// TwinCAT 3 PLC project PLC_Convert
// ProgramVersion: 3.1.4026.19
// libraries:
//   Tc2_Database, * (Beckhoff Automation GmbH)
//   Tc2_Drive, * (Beckhoff Automation GmbH)
//   Tc2_EtherCAT, * (Beckhoff Automation GmbH)
//   Tc2_IoFunctions, * (Beckhoff Automation GmbH)
//   Tc2_Math, * (Beckhoff Automation GmbH)
//   Tc2_MC2, * (Beckhoff Automation GmbH)
//   Tc2_MC2_Drive, * (Beckhoff Automation GmbH)
//   Tc2_SerialCom, * (Beckhoff Automation GmbH)
//   Tc2_Standard, * (Beckhoff Automation GmbH)
//   Tc2_System, * (Beckhoff Automation GmbH)
//   Tc2_SystemCX, * (Beckhoff Automation GmbH)
//   Tc2_TcpIp, * (Beckhoff Automation GmbH)
//   Tc2_Utilities, * (Beckhoff Automation GmbH)
//   Tc2_XmlDataSrv, * (Beckhoff Automation GmbH)
//   Tc3_EventLogger, * (Beckhoff Automation GmbH)
//   Tc3_Module, * (Beckhoff Automation GmbH)
//   TcUnit, * (www.tcunit.org)
// project tree:
//   / Control_Task.TcTTO, xFast_Task.TcTTO, Fast_Task.TcTTO, Accessory_Task.TcTTO, TcUnit_Task.TcTTO
//   Data types/METS/ADS Symobol/ E_SYMBOL_AccessState.TcDUT, E_SYMBOL_AdsStates.TcDUT, ST_SYMBOL_AddressInfo.TcDUT
//   Data types/METS/AI Codes And Validation/ E_CodeAI.TcDUT (not stored), E_CodeAIType.TcDUT, E_CodeType.TcDUT, ST_CodeInfo.TcDUT, ST_CodeValidation.TcDUT, ST_RejectItems.TcDUT, ST_RejectReasonsForCase.TcDUT, ST_RejectReasonsForOuter.TcDUT, ST_RejectReasonsForPack.TcDUT
//   Data types/METS/AI Codes And Validation/GS1_Standard/ E_GS1_CodeAIType.TcDUT, E_GS1_CodeLvl.TcDUT, ST_GS1_AI_Attributs.TcDUT, ST_GS1_AI_Definition.TcDUT, ST_GS1_CodeInfo.TcDUT, ST_GS1_CodeValidation.TcDUT, ST_GS1_Decode_AI.TcDUT
//   Data types/METS/Alarms/ E_MessageID.TcDUT, E_MessageType.TcDUT (not stored), ST_AlarmDB.TcDUT (not stored), ST_Alarms.TcDUT, ST_AlarmSettings.TcDUT, ST_AlarmsTable.TcDUT, ST_AlarmStatus.TcDUT, ST_ALARM_Aux.TcDUT
//   Data types/METS/Aliases/ T_CAC_Filename.TcDUT, T_CASE_Barcode.TcDUT, T_Char.TcDUT, T_CHM_Filename.TcDUT, T_CodeBATCH.TcDUT, T_CodeBRAND.TcDUT, T_CodeCRYPTO.TcDUT, T_CodeGTIN.TcDUT (not stored), T_CodeMRP.TcDUT, T_CodePIT.TcDUT, T_CodePO.TcDUT, T_CodePRODUCEDATE.TcDUT, T_CodeRSKU.TcDUT, T_CodeURL.TcDUT, T_DB_LongSTRING.TcDUT, T_FileExtension.TcDUT, T_FolderName.TcDUT, T_FolderPath.TcDUT (not stored), T_FSS_RejecCode.TcDUT, T_HMI_PACK_Barcode.TcDUT, T_ISO8601Time.TcDUT, T_LongSTRING.TcDUT, T_OAC_Filename.TcDUT, T_OCV_Filename.TcDUT, T_OHM_Filename.TcDUT, T_OUTER_Barcode.TcDUT, T_PACK_Barcode.TcDUT, T_PCM_Filename.TcDUT, T_PositiveINT.TcDUT (not stored), T_PositiveDINT.TcDUT (not stored), T_ProductDescription.TcDUT, T_RejectCode.TcDUT, T_TimeLog.TcDUT
//   Data types/METS/Case/CAC/ E_CAC_State.TcDUT, ST_CAC_Data.TcDUT
//   Data types/METS/Case/CHM/CHM Data Structure/GenericHierarchy/Case Item Structures/ ST_CaseContent.TcDUT (not stored), ST_CaseIdentity.TcDUT (not stored), ST_CaseItem.TcDUT (not stored)
//   Data types/METS/Case/CHM/CHM Data Structure/GenericHierarchy/Outer Item Structures/ ST_OuterContent.TcDUT (not stored), ST_OuterIdentity.TcDUT (not stored), ST_OuterItem.TcDUT (not stored)
//   Data types/METS/Case/CHM/CHM Data Structure/GenericHierarchy/Pack Item Structures/ ST_PackIdentity.TcDUT (not stored), ST_PackItem.TcDUT (not stored)
//   Data types/METS/Case/CHM/CHM Data Structure/GenericHierarchy/ ST_DefaultIdentity.TcDUT (not stored)
//   Data types/METS/Case/CHM/CHM Data Structure/ ST_Attributes.TcDUT, ST_CHM_GenericHierarchy.TcDUT (excluded from build), ST_GenericHierarchy.TcDUT, ST_MessageHeader.TcDUT
//   Data types/METS/Case/CHM/ E_CHM_GeneratorState.TcDUT, E_CHM_State.TcDUT, E_CHM_WriteMode.TcDUT (excluded from build), ST_CHM_Data.TcDUT
//   Data types/METS/Case/ E_CASE_State.TcDUT, ST_CasePackerInfo.TcDUT, ST_CASE_CaseQueue.TcDUT, ST_CASE_DefferOuter.TcDUT, ST_CASE_InfeedQueue.TcDUT (not stored), ST_CASE_OperationData.TcDUT
//   Data types/METS/Case/ORCA/ E_ORCA_State.TcDUT, ST_ORCA_BrandInfo.TcDUT, ST_ORCA_Data.TcDUT, ST_ORCA_Outers.TcDUT, ST_ORCA_ProductInfo.TcDUT, ST_ORCA_SiteInfo.TcDUT
//   Data types/METS/Device/CX Unit/Device/ E_CX_DeviceState.TcDUT (not stored)
//   Data types/METS/Device/CX Unit/EtherCAT/ E_CX_EtherCATState.TcDUT, ST_CX_EtherCATDeviceState.TcDUT, ST_CX_EtherCATMasterPNetState.TcDUT, ST_CX_EtherCATMasterState.TcDUT
//   Data types/METS/Device/CX Unit/EtherCAT/Terminal FBs/EBUS/ ST_EBUS_AnalogueDataIn.TcDUT (not stored), ST_EBUS_EtherCATState.TcDUT (not stored)
//   Data types/METS/Device/CX Unit/EtherCAT/Terminal FBs/KBUS/ E_KBUS_RegisterAccessState.TcDUT (not stored), ST_KBUS_AnalogueDataIn.TcDUT (not stored), ST_KBUS_AnalogueDataOut.TcDUT (not stored), ST_KBUS_KL1501DataIn.TcDUT (not stored), ST_KBUS_KL1501DataOut.TcDUT (not stored), ST_KBUS_KL5001Config.TcDUT (not stored)
//   Data types/METS/Device/CX Unit/EtherCAT/Terminal FBs/ ST_EtherCATSlaveInfo.TcDUT (not stored), ST_EtherCATStatus.TcDUT (not stored)
//   Data types/METS/Device/CX Unit/Network/ E_CX_NetworkInfoState.TcDUT (not stored), E_CX_SetAMSNetIDState.TcDUT (not stored), ST_CX_AdapterInfo.TcDUT, ST_CX_NetworkInfo.TcDUT
//   Data types/METS/Device/CX Unit/NOVRAM/ E_CX_NVDataCtrlState.TcDUT (not stored), E_CX_NVDataOpMode.TcDUT, E_CX_NVXMLState.TcDUT, ST_CX_AMSAddress.TcDUT, ST_CX_EL6080DataIn.TcDUT, ST_CX_EL6080DataOut.TcDUT, ST_CX_NVDataBlock.TcDUT
//   Data types/METS/Device/CX Unit/System/ E_CX_HWType.TcDUT (not stored), E_CX_State.TcDUT
//   Data types/METS/Device/Cylinders/ E_CYLINDER_Name.TcDUT, E_CYLINDER_Position.TcDUT (not stored), ST_CYLINDER_Config.TcDUT, ST_CYLINDER_Control.TcDUT, ST_CYLINDER_IN.TcDUT, ST_CYLINDER_OUT.TcDUT (not stored), ST_CYLINDER_Status.TcDUT, ST_CYLINDER_TagID.TcDUT
//   Data types/METS/Device/DB/ E_DB_ScanState.TcDUT, ST_DB_CACDataCtrl.TcDUT, ST_DB_OACDataCtrl.TcDUT (not stored), ST_DB_OCVDataCtrl.TcDUT (not stored)
//   Data types/METS/Device/DB/OLD/ ST_DBResult.TcDUT (excluded from build), ST_DB_CACCheckCtrl.TcDUT (excluded from build), ST_DB_Config.TcDUT, ST_DB_OACCheckCtrl.TcDUT (excluded from build), ST_DB_OCVCheckCtrl.TcDUT (excluded from build), ST_DB_PcvCheckCtrl.TcDUT (excluded from build), ST_DB_ReportDBCtrl.TcDUT, ST_DB_ReportResult.TcDUT
//   Data types/METS/Device/Drive/Analog/Config/ ST_AnalogDrive.TcDUT (not stored)
//   Data types/METS/Device/Drive/Analog/ ST_DriveCtrl.TcDUT, ST_PhtcCtrl.TcDUT (excluded from build)
//   Data types/METS/Device/Drive/MC2/Axis Control/ E_AXIS_MotionType.TcDUT (not stored), ST_AXIS_Control.TcDUT (not stored), ST_AXIS_IN.TcDUT (not stored), ST_AXIS_OUT.TcDUT (not stored), ST_AXIS_Status.TcDUT (not stored)
//   Data types/METS/Device/Drive/MC2/Config/ ST_AXIS_Config.TcDUT (not stored)
//   Data types/METS/Device/Drive/MC2/EtherCAT/AX5000 FBs/ ST_AX5000_TouchProbe.TcDUT (not stored)
//   Data types/METS/Device/Drive/MC2/EtherCAT/Encoder FBs/ ST_DeviceAddress.TcDUT (not stored)
//   Data types/METS/Device/Drive/MC2/ E_MC_Name.TcDUT
//   Data types/METS/Device/Drive/MC2/NC Axis/Cam/ E_CAM_Update.TcDUT (not stored)
//   Data types/METS/Device/Drive/MC2/NC Axis/ E_AXIS_CtrlState.TcDUT (not stored), E_TORQUE_Scaling.TcDUT (not stored), ST_AxisCtrlRamps.TcDUT (not stored), ST_DriveStatus.TcDUT (not stored), ST_LatchPosBuffer.TcDUT (not stored), ST_NC_EncDataIn.TcDUT (not stored), ST_NC_EncDataOut.TcDUT (not stored)
//   Data types/METS/Device/Drive/MC2/TempAxis/ ST_AxisHomeStruct.TcDUT (not stored) (excluded from build), ST_AxisMotionStruct.TcDUT (not stored) (excluded from build)
//   Data types/METS/Device/Drive/Profinet/Config/ ST_ProfinetDrive.TcDUT (not stored), ST_ProfinetMasterConfig.TcDUT (not stored)
//   Data types/METS/Device/Drive/Profinet/ E_DRIVE_Name.TcDUT (not stored), ST_PNetMasterStatus.TcDUT
//   Data types/METS/Device/Drive/Profinet/Parameters/ ST_DataPntAdr.TcDUT (not stored), ST_KeyPadDisplay.TcDUT (not stored), ST_Parameter.TcDUT (not stored), ST_ParameterControl.TcDUT (not stored), ST_Parameters.TcDUT (not stored), ST_Value.TcDUT (not stored)
//   Data types/METS/Device/Drive/Profinet/_G120/Drives/ E_DRIVE_DataType.TcDUT (not stored), ST_DRIVE_INPUT.TcDUT (not stored), ST_DRIVE_OUTPUT.TcDUT (not stored), ST_DRIVE_STATUS.TcDUT (not stored), ST_G120_ExtendedIn.TcDUT (not stored), ST_G120_ExtendedOut.TcDUT (not stored), ST_G120_IN.TcDUT (not stored), ST_G120_OUT.TcDUT (not stored), ST_G120_Status.TcDUT (not stored)
//   Data types/METS/Device/Drive/Profinet/_G120/ ST_G120_Control.TcDUT (not stored)
//   Data types/METS/Device/Encoders/CAMS/ ST_AFS60_Cam.TcDUT, ST_AFS60_CamHMi.TcDUT, ST_AFS60_Config.TcDUT, ST_AFS60_Status.TcDUT
//   Data types/METS/Device/Encoders/ E_ENOCDER_Name.TcDUT, ST_ENCODER_IN.TcDUT, ST_ENCODER_OUT.TcDUT (not stored), ST_ENCODER_Status.TcDUT
//   Data types/METS/Device/IO2 Controls/ E_IO2_InputSource.TcDUT (not stored), E_IO2_Type.TcDUT (not stored), ST_IO2_Diagnostic.TcDUT, ST_IO2_InputPLC.TcDUT, ST_IO2_OutputPLC.TcDUT
//   Data types/METS/Device/IO2 Controls/Input Ctrl/ ST_IO2_DoubleInputCtrl.TcDUT, ST_IO2_DoubleInputLockedCtrl.TcDUT, ST_IO2_SingleInputCtrl.TcDUT, ST_IO2_SingleInputLockedCtrl.TcDUT
//   Data types/METS/Device/IO2 Controls/Outpout Ctrl/ ST_IO2_OutputCtrl.TcDUT
//   Data types/METS/Device/Printers/ E_PRINTER_Name.TcDUT, E_PRINTER_State.TcDUT (not stored), ST_PRINTER_Config.TcDUT, ST_PRINTER_IN.TcDUT, ST_PRINTER_OUT.TcDUT, ST_PRINTER_Status.TcDUT
//   Data types/METS/Device/Scanner/ E_ClientSteps.TcDUT, E_DataExchaSteps.TcDUT, E_SCANNER_CodeType.TcDUT (not stored), E_SCANNER_DeviceType.TcDUT (not stored), E_SCANNER_Name.TcDUT, E_SCANNER_State.TcDUT (not stored), E_SCANNER_Vendor.TcDUT (not stored), ST_SCANNER.TcDUT, ST_SCANNER_ApplicationIdentifier.TcDUT, ST_SCANNER_CameraMap.TcDUT, ST_SCANNER_CodeData.TcDUT, ST_SCANNER_Config.TcDUT, ST_SCANNER_Evaluation.TcDUT, ST_SCANNER_ImageData.TcDUT, ST_SCANNER_ManualCtrl.TcDUT, ST_SCANNER_OpState.TcDUT, ST_SCANNER_Options.TcDUT, ST_SCANNER_Performance.TcDUT, ST_SCANNER_Statistics.TcDUT, ST_SCANNER_TriggerID.TcDUT
//   Data types/METS/Device/Scanner/Hand Scanner/ E_ConnectSteps.TcDUT, E_DataSequence.TcDUT (not stored), E_SCANNER_Baudrate.TcDUT, ST_SCANNER_HoneywellConfig.TcDUT, ST_SCANNER_HoneywellCtrl.TcDUT, ST_SCANNER_HoneywellStatus.TcDUT, ST_SCANNER_HostAck.TcDUT, ST_SCANNER_USBConfig.TcDUT
//   Data types/METS/Device/Scanner/NewModel/ ST_SCANNER_CtrlMapping.TcDUT, ST_SCANNER_Configuration.TcDUT, ST_SCANNER_Ctrl.TcDUT (not stored), ST_SCANNER_IN.TcDUT (not stored), ST_SCANNER_CtrlOptions.TcDUT (not stored) (excluded from build), ST_SCANNER_ManualStatus.TcDUT, ST_SCANNER_OUT.TcDUT, ST_SCANNER_Status.TcDUT
//   Data types/METS/Files/ E_FILE_CtrlState.TcDUT, E_FILE_DeleteOldFilesState.TcDUT, E_FILE_State.TcDUT, ST_FILE_WriteFileStatistic.TcDUT
//   Data types/METS/HMI/Device Manual Control/ ST_HMI_AxisCtrl.TcDUT, ST_HMI_CylinderCtrl.TcDUT, ST_HMI_G120Ctrl.TcDUT, ST_HMI_PrinterCtrl.TcDUT
//   Data types/METS/HMI/Device Status/ E_HMI_DriveStatus.TcDUT, ST_HMI_AxisStatus.TcDUT (not stored), ST_HMI_CylinderStatus.TcDUT, ST_HMI_G120Status.TcDUT, ST_HMI_HoneywellStatus.TcDUT, ST_HMI_PrinterStatus.TcDUT
//   Data types/METS/HMI/HMIQueue/ ST_HMI_CAC_Data.TcDUT, ST_HMI_CaseRejectCode.TcDUT, ST_HMI_CaseVerifiedCode.TcDUT (not stored), ST_HMI_CASE_CaseQueue.TcDUT (not stored), ST_HMI_InfeedQueue.TcDUT, ST_HMI_OAC_Data.TcDUT (not stored), ST_HMI_OCV_Data.TcDUT (not stored), ST_HMI_OuterStatus.TcDUT (not stored), ST_HMI_PACK_BufferStatus.TcDUT, ST_HMI_PLAS_Queue.TcDUT (not stored)
//   Data types/METS/HMI/ ST_HMI_BarGraph.TcDUT, ST_HMI_Buttons.TcDUT, ST_HMI_CSVStoreTable.TcDUT, ST_HMI_StationStatus.TcDUT (not stored), ST_HMI_Visualisation.TcDUT
//   Data types/METS/KPI/ ST_KPI_CasePackerSignals.TcDUT (not stored), ST_KPI_CodePos.TcDUT, ST_KPI_InspectionEfficency.TcDUT, ST_KPI_ItemsProduced.TcDUT, ST_KPI_OCVFile.TcDUT (not stored), ST_KPI_OutersProcessing.TcDUT, ST_KPI_OutersProduced.TcDUT
//   Data types/METS/LogData/ E_LOG_Handler.TcDUT, ST_LOG_Alarms.TcDUT (not stored), ST_LOG_EventData.TcDUT (not stored), ST_LOG_FileWriteError.TcDUT (not stored), ST_LOG_MachineState.TcDUT (not stored), ST_LOG_RejectReasons.TcDUT, ST_LOG_WriteImageData.TcDUT (not stored)
//   Data types/METS/NV Data/ ST_NOVRAM_METS_Cameras.TcDUT, ST_NOVRAM_METS_CaseInspactionLog.TcDUT (not stored), ST_NOVRAM_METS_DualInputs.TcDUT, ST_NOVRAM_METS_EventCounters.TcDUT, ST_NOVRAM_METS_Inspection.TcDUT
//   Data types/METS/Outers/ E_OUTER_AgrregationState.TcDUT, E_OUTER_State.TcDUT, ST_OUTER_Status.TcDUT
//   Data types/METS/Outers/OAC/ E_OAC_State.TcDUT, ST_OAC_Data.TcDUT
//   Data types/METS/Outers/SFLX/ E_SIDEFLEX_UnitType.TcDUT, ST_SIDEFLEX_Offset.TcDUT, ST_SIDEFLEX_ProcessData.TcDUT
//   Data types/METS/Packs/ E_OCV_CheckMode.TcDUT, E_OCV_State.TcDUT, E_PACK_FilledInStatus.TcDUT, E_PACK_ReadStep.TcDUT, E_PACK_State.TcDUT, ST_PACK_CodeBuffer.TcDUT, ST_PACK_CodeStatus.TcDUT, ST_PACK_ConfirmationQueue.TcDUT, ST_PACK_Data.TcDUT, ST_PACK_DuplicatesCheck.TcDUT, ST_PACK_InfeedQueue.TcDUT, ST_PACK_InTransferQueue.TcDUT, ST_PACK_LastFilledCodes.TcDUT, ST_PACK_TriggerOffset.TcDUT
//   Data types/METS/Packs/_Lab/ ST_LAB_PackData.TcDUT, ST_LAB_OuterData.TcDUT
//   Data types/METS/PCM/ E_PCM_State.TcDUT, ST_PCM_Data.TcDUT, ST_PCM_Status.TcDUT (not stored)
//   Data types/METS/PCM/PCM_Hierarchy/ProductInformation/Product/ ST_HierarchyData.TcDUT (not stored), ST_HierarchyDataList.TcDUT (not stored)
//   Data types/METS/PCM/PCM_Hierarchy/ProductInformation/Settings/ ST_ToleranceThresholdCS.TcDUT (not stored), ST_ToleranceThresholdOUT.TcDUT (not stored), ST_ToleranceThresholdPK.TcDUT (not stored)
//   Data types/METS/PCM/PCM_Hierarchy/ProductInformation/ ST_PCMProduct.TcDUT, ST_PCMSettings.TcDUT
//   Data types/METS/PCM/PCM_Hierarchy/ ST_PCMMessageHeader.TcDUT, ST_ProductInformation.TcDUT
//   Data types/METS/String Processing/ E_STRING_ExtrMode.TcDUT
//   Data types/METS/System/ E_SYSTEM_CTState.TcDUT, E_SYSTEM_HandScannerBaudrate.TcDUT, E_SYSTEM_ItemType.TcDUT, E_SYSTEM_MachineState.TcDUT (not stored), E_SYSTEM_MaintainFolders.TcDUT (not stored), E_SYSTEM_OSType.TcDUT, ST_SYSTEM_Config.TcDUT, ST_SYSTEM_DateTime.TcDUT, ST_SYSTEM_DeviceState.TcDUT, ST_SYSTEM_Door.TcDUT, ST_SYSTEM_MachineID.TcDUT, ST_SYSTEM_MachineMode.TcDUT, ST_SYSTEM_MachineState.TcDUT, ST_SYSTEM_ProductionLine.TcDUT, ST_SYSTEM_SafetyStatus.TcDUT, ST_SYSTEM_SoftwareVersion.TcDUT
//   Data types/METS/System/Status/ ST_SYSTEM_ArchiveDBStatus.TcDUT, ST_SYSTEM_ReportingDBStatus.TcDUT (not stored), ST_SYSTEM_BridgeStatus.TcDUT (not stored), ST_SYSTEM_LoggerStatus.TcDUT, ST_SYSTEM_MachineStatus.TcDUT (not stored)
//   Data types/METS/System/System Modes/ E_SYSTEM_AutomationMode.TcDUT, E_SYSTEM_OuterAggregationMode.TcDUT, E_SYSTEM_PackAggregationMode.TcDUT (not stored)
//   Data types/METS/TCPIP Address/ E_TCPIP_State.TcDUT, ST_TCPIP_AddressPort.TcDUT
//   Data types/METS/XML Processing/ E_XML_CtrlState.TcDUT, E_XML_GeneratorState.TcDUT, E_XML_WritingMode.TcDUT
//   Data types/METS/_StationOperational/C715 Tempalate Example/ E_04_ElevatorState_C715.TcDUT, E_Axis_C715.TcDUT, E_Cylinder_C715.TcDUT, ST_04_ElevatorSeq_C715.TcDUT, ST_BundleTrackingRegister_C715.TcDUT, ST_CommonStationConfig_C715.TcDUT
//   Data types/METS/_StationOperational/ E_00_StationStateTemplate.TcDUT, ST_00_StationStructTemplate.TcDUT
//   Data types/METS/_StationOperational/Manual Machine/ E_OuterPrintStationState.TcDUT, ST_OuterPrintStationStruct.TcDUT (not stored)
//   Data types/METS/_StationOperational/SeqCtrl/ ST_STATION_Requests.TcDUT, ST_STATION_Status.TcDUT
//   POUs/METS/Common LIB/04_CASE LIB/Case FBs/FinaliseCaseData/ FB_CASE_DuplicatCheck.TcPOU (not stored), FB_CASE_DuplicateUpdateToDB.TcPOU (not stored), FB_CASE_FinaliseData.TcPOU (not stored), FB_CASE_InitialiseData.TcPOU (not stored), FB_CASE_MovePackerToCase.TcPOU (not stored), FB_CASE_ValidateContent.TcPOU (not stored)
//   POUs/METS/Common LIB/07_DEVICE LIB/CommonCX FBs %28Hardware%29/EtherCAT FBs/Obsolete/ FB_CX_EtherCATDevState.TcPOU (not stored) (excluded from build), FB_CX_EtherCATSlaveDiag.TcPOU (not stored) (excluded from build), FB_EtherCAT_Status.TcPOU (not stored) (excluded from build)
//   POUs/METS/Common LIB/07_DEVICE LIB/CommonCX FBs %28Hardware%29/Non-Volatile Data FBs/Obsolete/ FB_CX_NVData_BinaryFile_4K.TcPOU (not stored) (excluded from build), FB_CX_NVData_EL6080_1K.TcPOU (not stored) (excluded from build), FB_CX_NVData_Generic1K.TcPOU (not stored) (excluded from build)
//   POUs/METS/Common LIB/08_SOFTWARE LIB/AI Codes And Validation FBs/ F_CODE_GetItemAI.TcPOU, FB_CODE_ClearCodeInfo.TcPOU, FB_CODE_ValidateExplicitCode.TcPOU (not stored), F_CODE_AssignValToString.TcPOU, F_CODE_AssignValToStringWithPrefix.TcPOU (not stored), F_CODE_GetItem.TcPOU
//   POUs/METS/Common LIB/09_SYSTEM LIB/Alarm/ FB_ALARM_Handler.TcPOU (not stored), FB_ALARM_GroupManagment.TcPOU (not stored), FB_ALARM_LogTable.TcPOU (not stored), FB_ALARM_Message.TcPOU (not stored) (excluded from build), FB_ALARM_OutputDB.TcPOU (not stored) (excluded from build), F_ALARM_SetDefinition.TcPOU (not stored)
//   POUs/METS/Common LIB/09_SYSTEM LIB/ FB_SYSTEM_CoreFolders.TcPOU, FB_SYSTEM_CorePaths.TcPOU, FB_SYSTEM_AverageTimeDiff.TcPOU, FB_SYSTEM_BarcodeType.TcPOU, FB_SYSTEM_DateTime.TcPOU, FB_SYSTEM_HardwareOS.TcPOU, FB_SYSTEM_MachineState.TcPOU, FB_SYSTEM_ProdMonitor.TcPOU, FB_SYSTEM_SearchBarcode.TcPOU, FB_SYSTEM_SeqControl.TcPOU, FB_SYSTEM_ShiftMonitor.TcPOU, FB_SYSTEM_TaskInfo.TcPOU, FB_SYSTEM_ValidateSettings.TcPOU
//   POUs/METS/METS General/01 Control Task %28Process%29/ C13_CheckDuplicatesCACData.TcPOU (not stored), C01_System.TcPOU (not stored), C02_PCM.TcPOU (not stored), C03_AlarmMessageControl.TcPOU (not stored), C04_ContolButtons.TcPOU (not stored), C05_MachineStatus.TcPOU (not stored), C06_TowerLamps.TcPOU (not stored), C07_EtherCATDiagnostic.TcPOU (not stored), C08_PulseGenerator.TcPOU (not stored), C09_MaintainFolders.TcPOU (not stored), C10_PackControlOCVData.TcPOU (not stored), C11_OuterControlOACData.TcPOU (not stored), C12_InfeedConvAddOACData.TcPOU (not stored), C20_ProfinetDrivesCtrl.TcPOU (not stored), C21_CamerasCtrl.TcPOU (not stored), C25_MC2AxisDriversCtrl.TcPOU (not stored), C30_DiagnosticHMI.TcPOU (not stored)
//   POUs/METS/METS General/02 Accessory Task %28External%29/ A10_LAB_Duplicat.TcPOU (not stored) (excluded from build), A04_StartupWebHMI.TcPOU (not stored), A01_StartupBridge.TcPOU (not stored), A07_BargraphHMI.TcPOU (not stored), A06_AuxInterface.TcPOU (not stored), A08_CodeInfoCtrl.TcPOU (not stored), A09_CurrentStatistic.TcPOU (not stored), A03_StartupLogger.TcPOU (not stored), A02_StartupArchiveDB.TcPOU (not stored), A05_StartupReportingDB.TcPOU (not stored) (excluded from build)
//   POUs/TcUnit/FB_CASE_ValidateContentTests/ FB_CASE_ValidateContentTests.TcPOU, PRG_CASE_ValidateContentManual.TcPOU
//   POUs/_Exclude/ F13_CaseContentValidation_ORG.TcPOU (excluded from build), FB_CASE_FinaliseCaseData.TcPOU (excluded from build), FB_CASE_ValidateCaseContent.TcPOU (excluded from build), FB_SYSTEM_CheckOS.TcPOU (excluded from build), FB_SYSTEM_CreateFolders.TcPOU (excluded from build), C09_MaintainFolders_OLD.TcPOU (excluded from build), C09_MaintainFolders_ORG.TcPOU (excluded from build), F15_CaseControlCACData_ORG.TcPOU (excluded from build), F21_ContentHandScanner_ORG.TcPOU (excluded from build), F41_EventLoggerPT.TcPOU (excluded from build), F42_EventLoggerML.TcPOU (excluded from build), F43_EventLoggerOT.TcPOU (excluded from build), F44_EventLoggerCT.TcPOU (excluded from build), FB_CASE_AddOACDataLoop.TcPOU (excluded from build), FB_CASE_ShiftCaseQueue_ORG.TcPOU (excluded from build), FB_CHM_ClearArchive.TcPOU (excluded from build), FB_CX_NVData_NOVRAM_4K.TcPOU (excluded from build), FB_MemoryMonitor_32K.TcPOU (excluded from build), FB_MemoryMonitor_4K.TcPOU (excluded from build), FB_OUTER_CompleteDataFromConfirmation.TcPOU (excluded from build), FB_OUTER_CompleteDataFromOCV.TcPOU (excluded from build), FB_OUTER_RefeedOCVFilesWtihError.TcPOU (excluded from build), FB_OUTER_RepairOCVContent.TcPOU (excluded from build), FB_OUTER_WriteOACFileLoop.TcPOU (excluded from build), FB_PACK_DuplicatesPackCodes.TcPOU (excluded from build), FB_PACK_ValidateOCVContent.TcPOU (excluded from build), FB_PACK_WriteOCVFileLoop_v3.TcPOU (excluded from build), FB_T03_MoveDataToOCVStatus_ORG.TcPOU (excluded from build), F_ALARM_SetDefinition_ORG.TcPOU (excluded from build), PRG_LARS_ValidationAsConfirmation_ORG.TcPOU (excluded from build), TestBlock_Check3.TcPOU (excluded from build), TestBlock_Check4.TcPOU (excluded from build)
//   Global Variables/ gMessage.TcGVL, gConstants.TcGVL (not stored), gHMI.TcGVL, CodeAI.TcGVL (not stored), gIOFiltered.TcGVL, gPersistent.TcGVL, gNovRAM.TcGVL
//   Global Variables/InputsOutputsDT/ gCamDevice.TcGVL, IOVarDT_S.TcGVL, IOVarDT_H.TcGVL, _Labs.TcGVL
//   Global Variables/InputsOutputs_CML/ IOVariablesCX_CML.TcGVL (excluded from build), IOVariablesEUCA_CML.TcGVL (excluded from build), IOVariablesPACAN_CML.TcGVL (excluded from build), IOVariablesPAOL_CML.TcGVL (excluded from build), IOVariablesPLAS_CML.TcGVL (excluded from build)
//   Global Variables/InputsOutputs_OC/ IOVariablesCX_OC.TcGVL (excluded from build), IOVariablesEUCA_OC.TcGVL (excluded from build), IOVariablesPAOL_OC.TcGVL (excluded from build), IOVariablesPLAS_OC.TcGVL (excluded from build)
//   Global Variables/InputsOutputs_SFLX/ IOVariablesCX_SFLX.TcGVL (excluded from build), IOVariablesEUCA_SFLX.TcGVL (excluded from build), IOVariablesPAOL_SFLX.TcGVL (excluded from build), IOVariablesPLAS_SFLX.TcGVL (excluded from build)
//   Global Variables/METS/ gDevice.TcGVL, gProcess.TcGVL
//   Global Variables/_VERSION/ _VERSION_CONTROL.TcGVL
//   POUs/METS/Common LIB/01_PACK LIB/OCV FBs/ FB_OCV_FindDB.TcPOU
//   POUs/METS/Common LIB/01_PACK LIB/Pack FBs/ FB_PACK_DuplicatesPackCodesDB.TcPOU, FB_PACK_MoveOuterStatusArray.TcPOU, FB_PACK_WriteOCVLoopDB.TcPOU
//   POUs/METS/Common LIB/01_PACK LIB/Pack FBs/PAOL/2CAM %28METS ONE%29/ FB_2CAM_AddPackCodes.TcPOU (not stored), FB_2CAM_CameraBoxRead.TcPOU (not stored), FB_2CAM_CameraSequenceNo.TcPOU (not stored), FB_2CAM_PackScanners2x5Packs.TcPOU (not stored), FB_2CAM_SelectCameraMap.TcPOU (not stored)
//   POUs/METS/Common LIB/01_PACK LIB/Pack FBs/PAOL/3CAM %28LIGHTBOX%29/ FB_3CAM_AddPackCodes.TcPOU (not stored), FB_3CAM_CameraBoxRead.TcPOU (not stored), FB_3CAM_CameraSequenceNo.TcPOU (not stored), FB_3CAM_PackScanners2x5Packs.TcPOU (not stored), FB_3CAM_PackScanners3x4Packs.TcPOU (not stored), FB_3CAM_PackScanners4x3Packs.TcPOU (not stored), FB_3CAM_SelectCameraMap.TcPOU (not stored)
//   POUs/METS/Common LIB/01_PACK LIB/Pack FBs/PAOL/ FB_PAOL_AddNewTriggerID.TcPOU (not stored), FB_PAOL_InfeedCamerasSync.TcPOU (not stored)
//   POUs/METS/Common LIB/01_PACK LIB/Pack FBs/PLAS/ FB_PLAS_AddInterimCodeToQ.TcPOU (not stored), FB_PLAS_AddNewTriggerID.TcPOU (not stored), FB_PLAS_FillInPackData.TcPOU (not stored), FB_PLAS_FillInPackDataWithCodeType.TcPOU (not stored) (excluded from build), FB_PLAS_InterimShiftQueue.TcPOU (not stored), FB_PLAS_MasterListAddToQueue.TcPOU (not stored), FB_PLAS_MasterListFillInPack.TcPOU (not stored), FB_PLAS_MasterListFillInPackRev.TcPOU (not stored), FB_PLAS_MasterListShiftQueue.TcPOU (not stored)
//   POUs/METS/Common LIB/01_PACK LIB/Pack FBs/PLAS/Type 01 %28CW - GD%29/ FB_T01_Add2PackToInfeedQ.TcPOU (not stored), FB_T01_CompleteOCV.TcPOU (not stored), FB_T01_MovePackToStacker.TcPOU (not stored)
//   POUs/METS/Common LIB/01_PACK LIB/Pack FBs/PLAS/Type 02 %28NCW - GD%29/ FB_T02_Add2PackToInfeedQ.TcPOU (not stored), FB_T02_CompleteOCV.TcPOU (not stored), FB_T02_MovePackToStacker.TcPOU (not stored), FB_T02_PackScanners2x5Packs.TcPOU (not stored) (excluded from build)
//   POUs/METS/Common LIB/01_PACK LIB/Pack FBs/PLAS/Type 03 %28NCW - FOCKE%29/ FB_T03_AddMultiPackToInfeedQ.TcPOU (not stored), FB_T03_CompleteOCV.TcPOU (not stored), FB_T03_MoveDataToOCVStatus.TcPOU (not stored), FB_T03_PackScanners2x5Packs.TcPOU (not stored) (excluded from build), FB_T03_PackScanners5x2Packs.TcPOU (not stored) (excluded from build)
//   POUs/METS/Common LIB/01_PACK LIB/Pack FBs/PLAS/Type 04 %28NCW - FOCKE H%29/ FB_T04_AddMultiPackToInfeedQ.TcPOU (not stored), FB_T04_CompleteOCV.TcPOU (not stored), FB_T04_MoveDataToOCVStatus.TcPOU (not stored)
//   POUs/METS/Common LIB/01_PACK LIB/Pack Functions/ F_PACK_GetRejectReasonFSS.TcPOU, F_PACK_HexToPackCode.TcPOU, F_PACK_ProgNumberMap.TcPOU, F_PACK_ValidateCodeASCII.TcPOU, F_PACK_ValidateHexName.TcPOU, F_PACK_ValidateTimeStamp.TcPOU
//   POUs/METS/Common LIB/02_OUTER LIB/OAC FBs/ FB_OAC_FindDB.TcPOU
//   POUs/METS/Common LIB/02_OUTER LIB/Outer FBs/Complete OCV/ FB_OUTER_CompleteDataFromDB_DoubleCam.TcPOU (not stored), FB_OUTER_CompleteDataFromDB_SingleCam.TcPOU (not stored), FB_OUTER_CompleteDataFromQueue_NoCam.TcPOU (not stored)
//   POUs/METS/Common LIB/02_OUTER LIB/Outer FBs/ FB_OUTER_ArchiveInvalidOuters.TcPOU, FB_OUTER_CheckDuplicateStatus.TcPOU, FB_OUTER_FindErrorOuter.TcPOU, FB_OUTER_InterimCameraOut.TcPOU, FB_OUTER_MasterListUpdate.TcPOU, FB_OUTER_MoveOuterStatus.TcPOU, FB_OUTER_RepairOCVContentDB.TcPOU, FB_OUTER_RestoreOCVDataFromStruct.TcPOU, FB_OUTER_ShiftConfimrCodeQ.TcPOU, FB_OUTER_ValidateOuterForReject.TcPOU, FB_OUTER_ValidationCameraOut.TcPOU, FB_OUTER_WriteErrorTable.TcPOU, FB_OUTER_WriteOACLoopDB.TcPOU
//   POUs/METS/Common LIB/02_OUTER LIB/Outer Functions/ F_OUTER_BarcodeToHex.TcPOU, F_OUTER_GetRejectReasonFSS.TcPOU, F_OUTER_HexToBarcode.TcPOU, F_OUTER_ProgNumberMap.TcPOU
//   POUs/METS/Common LIB/04_CASE LIB/Case FBs/ FB_CASE_AddOACDataDBLoop.TcPOU, FB_CASE_AddOuterToInfeedQ.TcPOU, FB_CASE_AddVerifiedCaseBarcode.TcPOU, FB_CASE_BiuldPackerLogString.TcPOU, FB_CASE_FindAndDeleteOuter.TcPOU, FB_CASE_FindCaseInQueue.TcPOU, FB_CASE_LastRowPoisitionBuffer_v2.TcPOU, FB_CASE_MasterListControl.TcPOU, FB_CASE_MoveFailedCAC.TcPOU, FB_CASE_MoveOutersRowToPacker.TcPOU, FB_CASE_MoveVerifiedCAC.TcPOU, FB_CASE_RestoreDataControl.TcPOU, FB_CASE_ShiftCaseQueue.TcPOU, FB_CASE_ShiftPackerQueue.TcPOU, FB_CASE_ValidatePrintCACData.TcPOU
//   POUs/METS/Common LIB/04_CASE LIB/Case Functons/ F_CASE_AddAIBrackets.TcPOU, F_CASE_BarcodeToCACFilename.TcPOU, F_CASE_ClearCACData.TcPOU, F_CASE_ClearCaseQueue.TcPOU, F_CASE_ClearCurrentPackerData.TcPOU, F_CASE_ClearFailedCaseQueue.TcPOU, F_CASE_ClearInfeedQueue.TcPOU, F_CASE_ClearPackerQueue.TcPOU, F_CASE_GetRejectReasonFSS.TcPOU, F_CASE_GetSKUFromHex.TcPOU (not stored)
//   POUs/METS/Common LIB/04_CASE LIB/Files FBs/CAC FBs/ FB_CAC_RestoreDataFromDB.TcPOU (not stored), FB_CAC_WriteHierachyToDB.TcPOU (not stored)
//   POUs/METS/Common LIB/04_CASE LIB/Files FBs/CHM FBs/ FB_CHM_FindFile.TcPOU (not stored), FB_CHM_MoveToArchive.TcPOU (not stored), FB_CHM_SaveFLG_File.TcPOU (not stored), FB_CHM_WriteFSS3Files.TcPOU (not stored)
//   POUs/METS/Common LIB/04_CASE LIB/Files FBs/CHM FBs/FSS3/ FB_CHM_PopulateDataForFSS3.TcPOU (not stored)
//   POUs/METS/Common LIB/04_CASE LIB/Files FBs/CHM FBs/FSS3/v4/ FB_CHM_BiuldXMLImige_v4.TcPOU (not stored), FB_CHM_HierachyFileGenerator.TcPOU (not stored)
//   POUs/METS/Common LIB/06_KPI LIB/ClearStatistic/ FB_KPI_ClearCameraInspection.TcPOU, FB_KPI_ClearExtCSStatistic.TcPOU, FB_KPI_ClearExtOUTStatistic.TcPOU, FB_KPI_ClearExtPKStatistic.TcPOU, FB_KPI_ClearFrontScreenStatistic.TcPOU, FB_KPI_ClearGeneraStatistic.TcPOU, FB_KPI_ClearInspectionStatistic.TcPOU, FB_KPI_ClearPackOuterInspection.TcPOU (excluded from build)
//   POUs/METS/Common LIB/06_KPI LIB/ItemEfficiency/ FB_KPI_CaseEfficiency.TcPOU, FB_KPI_InterimEfficiency.TcPOU (excluded from build), FB_KPI_OutersEfficiency.TcPOU, FB_KPI_PackEfficiency.TcPOU
//   POUs/METS/Common LIB/06_KPI LIB/ItemEfficiency/Generic/ FB_KPI_GenericEfficiency.TcPOU (not stored)
//   POUs/METS/Common LIB/06_KPI LIB/RejectCounters/ FB_KPI_CaseLevelCounter.TcPOU, FB_KPI_OuterLevelCounter.TcPOU, FB_KPI_PackLevelCounter.TcPOU
//   POUs/METS/Common LIB/07_DEVICE LIB/CommonCX FBs %28Hardware%29/CXDisplay FBs/ FB_CX_CX1100Display.TcPOU (not stored) (excluded from build), FB_CX_CX2100Display.TcPOU (not stored) (excluded from build)
//   POUs/METS/Common LIB/07_DEVICE LIB/CommonCX FBs %28Hardware%29/EtherCAT FBs/ FB_CX_EtherCATStatus.TcPOU (not stored)
//   POUs/METS/Common LIB/07_DEVICE LIB/CommonCX FBs %28Hardware%29/ FB_CX_GetDeviceID.TcPOU (not stored)
//   POUs/METS/Common LIB/07_DEVICE LIB/CommonCX FBs %28Hardware%29/Network FBs/ FB_CX_NetworkInfo.TcPOU (not stored), F_CX_LocalIPAddr.TcPOU (not stored)
//   POUs/METS/Common LIB/07_DEVICE LIB/CommonCX FBs %28Hardware%29/Non-Volatile Data FBs/ FB_CX_NVData_NOVRAM.TcPOU (not stored), FB_CX_NVData_XMLFile.TcPOU (not stored)
//   POUs/METS/Common LIB/07_DEVICE LIB/CommonCX FBs %28Hardware%29/Non-Volatile Data FBs/Internal FBs/ FB_CX_NVData_Transfer.TcPOU (not stored), F_ASCIIWordToByteValue.TcPOU (not stored), F_ByteValueToASCIIWord.TcPOU (not stored)
//   POUs/METS/Common LIB/07_DEVICE LIB/CommonCX FBs %28Hardware%29/Terminal FBs/EBUS/ FB_EBUS_020mASensor.TcPOU (not stored), FB_EBUS_10VSensor.TcPOU (not stored), FB_EBUS_420mASensor.TcPOU (not stored), FB_EBUS_TempSensor.TcPOU (not stored)
//   POUs/METS/Common LIB/07_DEVICE LIB/Cylinders/ FB_Cylinder.TcPOU, FB_CylinderWithMeasur.TcPOU (excluded from build)
//   POUs/METS/Common LIB/07_DEVICE LIB/DB Control/Connection Parameters/ FB_DB_CreateConnectionParams.TcPOU (not stored) (excluded from build)
//   POUs/METS/Common LIB/07_DEVICE LIB/DB Control/_internal/ FB_DBStoredProceduresRecordArrayLoop.TcPOU (not stored) (excluded from build)
//   POUs/METS/Common LIB/07_DEVICE LIB/Door/ FB_DOOR_RejectCtrl.TcPOU (excluded from build)
//   POUs/METS/Common LIB/07_DEVICE LIB/Drives/AX5000 FBs/ FB_MC2_AX5000AxisCtrl.TcPOU (not stored), FB_MC2_AX5000LatchPulse.TcPOU (not stored), FB_MC2_AX5000LatchPulseWidth.TcPOU (not stored), FB_MC2_AX5000Torque.TcPOU (not stored), FB_MC2_AX5000TorqueCtrl.TcPOU (not stored)
//   POUs/METS/Common LIB/07_DEVICE LIB/Drives/AX5000 FBs/Internal FBs/ FB_MC2_AX5000Status.TcPOU (not stored)
//   POUs/METS/Common LIB/07_DEVICE LIB/Drives/Axis Ctrl FBs/ FB_MC2_AbsCtrl.TcPOU (not stored), FB_MC2_BasicAxisCtrl.TcPOU (not stored), FB_MC2_CamCtrl.TcPOU (not stored) (excluded from build), FB_MC2_DigLockCtrl.TcPOU (not stored) (excluded from build), FB_MC2_RelCtrl.TcPOU (not stored), FB_MC2_VeloCtrl.TcPOU (not stored)
//   POUs/METS/Common LIB/07_DEVICE LIB/Drives/Conveyors/ FB_ACTransferControl.TcPOU (not stored) (excluded from build), FB_ConveyorControl.TcPOU (not stored) (excluded from build), FB_ConveyorCtrl.TcPOU (not stored) (excluded from build), FB_DriveAnalog.TcPOU (not stored) (excluded from build), FB_SeparatorCtrl.TcPOU (not stored) (excluded from build)
//   POUs/METS/Common LIB/07_DEVICE LIB/Drives/EL7201 FBs/ FB_MC2_EL7201AxisCtrl.TcPOU (not stored), FB_MC2_EL7201Torque.TcPOU (not stored), FB_MC2_EL7201TorqueCtrl.TcPOU (not stored)
//   POUs/METS/Common LIB/07_DEVICE LIB/Drives/EL7201 FBs/Internal FBs/ FB_MC2_EL7201Status.TcPOU (not stored)
//   POUs/METS/Common LIB/07_DEVICE LIB/Drives/Profinet Drives/Drive Control/ FB_DRIVE_SetControl.TcPOU (not stored), FB_G120Simple_V001.TcPOU (not stored), FB_ResetPulseGenerator.TcPOU (not stored), FB_SafetyResetSequencer.TcPOU (not stored) (excluded from build), F_DRIVE_GetStatus.TcPOU (not stored)
//   POUs/METS/Common LIB/07_DEVICE LIB/Drives/Profinet Drives/Drive Parameters/Function Blocks/ FB_ParameterDisplayWrapper.TcPOU (not stored) (excluded from build), FB_ReadDriveParametersPNET.TcPOU (not stored) (excluded from build), FB_WriteDriveParametersPNET.TcPOU (not stored) (excluded from build)
//   POUs/METS/Common LIB/07_DEVICE LIB/Drives/Profinet Drives/Drive Parameters/Functions/ FC_InitG120ReadPara.TcPOU (not stored) (excluded from build), FC_InitG120ReadWritePara.TcPOU (not stored) (excluded from build), FC_ReturnPointerForType.TcPOU (not stored) (excluded from build), FC_Round.TcPOU (not stored) (excluded from build)
//   POUs/METS/Common LIB/07_DEVICE LIB/Encoders/ FB_ENCODER_AbsValueToPos.TcPOU, FB_ENCODER_CamCtrl.TcPOU (excluded from build), FB_ENCODER_SingleTurn.TcPOU
//   POUs/METS/Common LIB/07_DEVICE LIB/IO2 Controls/ FB_IO2_DoubleInputCtrl.TcPOU, FB_IO2_DoubleInputLockCtrl.TcPOU, FB_IO2_ForceOutputs.TcPOU, FB_IO2_OutputCtrl.TcPOU, FB_IO2_SingleInputCtrl.TcPOU, FB_IO2_SingleInputLockCtrl.TcPOU, FB_IO_ForceOutputs.TcPOU (excluded from build)
//   POUs/METS/Common LIB/07_DEVICE LIB/Printer FBs/Domino/ FB_PRINTER_DominoMSeriesCtrl.TcPOU (not stored), FB_PRINTER_SelectCommand.TcPOU (not stored), F_PRINTER_Outer5Fields.TcPOU (not stored)
//   POUs/METS/Common LIB/07_DEVICE LIB/Scanner FBs %28Camera%29/Additional FBs/ FB_SCANNER_CheckOS.TcPOU (not stored), FB_SCANNER_CodeDiagnostic.TcPOU (not stored) (excluded from build), FB_SCANNER_DiagnosticLog.TcPOU (not stored), FB_SCANNER_DecodeGS1.TcPOU (not stored), FB_SCANNER_Evaluation.TcPOU (not stored), FB_SCANNER_KeyenceBrowse.TcPOU (not stored), FB_SCANNER_KeyenceDecodeImageData.TcPOU (not stored), FB_SCANNER_MICROSCANBrowse.TcPOU (not stored), FB_SCANNER_MicroscanDecodeImageData.TcPOU (not stored), FB_SCANNER_MV4x0Browse.TcPOU (not stored), FB_SCANNER_MVxDecodeImageData.TcPOU (not stored), FB_SCANNER_OmronDecodeImageData.TcPOU (not stored), FB_SCANNER_SiemensMV4x0Ctrl_Server.TcPOU (not stored) (excluded from build), F_SCANNER_CodeMaxLenghtCheck.TcPOU (not stored), F_SCANNER_FindCodeType.TcPOU (not stored), F_SCANNER_Keyence_SymbolID_To_CodeType.TcPOU (not stored), F_SCANNER_LightingIntensity.TcPOU (not stored), F_SCANNER_MV4x0Options.TcPOU (not stored) (excluded from build), F_SCANNER_OpState.TcPOU (not stored), F_SCANNER_RemoveAIBrackets.TcPOU (not stored), F_SCANNER_TriggerID.TcPOU (not stored)
//   POUs/METS/Common LIB/07_DEVICE LIB/Scanner FBs %28Camera%29/Cameras/ FB_SCANNER_CameraSelect.TcPOU (not stored), FB_SCANNER_MicroScan.TcPOU (not stored), FB_SCANNER_OmronFJCtrl.TcPOU (not stored), FB_SCANNER_SiemensMV4x0Ctrl.TcPOU (not stored)
//   POUs/METS/Common LIB/07_DEVICE LIB/Scanner FBs %28Camera%29/NewModel/ FB_SCANNER_CameraSelectExt.TcPOU (not stored), FB_SCANNER_KeyenceExt.TcPOU (not stored), FB_SCANNER_OmronExt.TcPOU (not stored), FB_SCANNER_SiemensExt.TcPOU (not stored)
//   POUs/METS/Common LIB/07_DEVICE LIB/Scanner FBs %28Camera%29/SerialScanners/ FB_HandScannerAddress.TcPOU (not stored), FB_HandScannerCtrl.TcPOU (not stored), FB_SCANNER_BaudrateMonitor.TcPOU (not stored), FB_SCANNER_HoneyWellControl.TcPOU (not stored), FB_SCANNER_SerialCom_v2.TcPOU (not stored)
//   POUs/METS/Common LIB/08_SOFTWARE LIB/AI GS1 Codes And Validation FBs/ FB_GS1_ClearCodeInfo.TcPOU, FB_GS1_ValidateExplicitCode.TcPOU, F_GS1_GetItem.TcPOU
//   POUs/METS/Common LIB/08_SOFTWARE LIB/Cog Checker FB/CogChecker/ FB_COG_Chek.TcPOU (not stored) (excluded from build), F_CogCheck.TcPOU (not stored) (excluded from build), F_MulMod.TcPOU (not stored) (excluded from build)
//   POUs/METS/Common LIB/08_SOFTWARE LIB/Cog Checker FB/ FB_CogCorrection.TcPOU (excluded from build), F_COG_Checker.TcPOU (excluded from build)
//   POUs/METS/Common LIB/08_SOFTWARE LIB/Counter FBs/ FB_ChangeStateTrig.TcPOU, FB_CTD32.TcPOU, FB_CTU16.TcPOU, FB_CTU32.TcPOU, FB_Incrementer.TcPOU, FB_InWindow.TcPOU
//   POUs/METS/Common LIB/08_SOFTWARE LIB/Debug/ FB_DEBUG_CounterArray.TcPOU
//   POUs/METS/Common LIB/08_SOFTWARE LIB/File FBs/ FB_FILE_ApendWriteByByte.TcPOU, FB_FILE_Compare.TcPOU, FB_FILE_Copy.TcPOU, FB_FILE_CopyByByte.TcPOU, FB_FILE_Delete.TcPOU, FB_FILE_DeleteOldFiles.TcPOU, FB_FILE_GetFileInfo.TcPOU, FB_FILE_GetFileList.TcPOU, FB_FILE_Move.TcPOU, FB_FILE_MoveWithDate.TcPOU, FB_FILE_ReadByByte.TcPOU, FB_FILE_Rename.TcPOU, FB_FILE_WriteByByte.TcPOU, F_FILE_AppendStringToFileName.TcPOU, F_FILE_CompareFileTime.TcPOU, F_FILE_FileTimeToULarge.TcPOU, F_FILE_SetFileExtension.TcPOU, F_FILE_SplitFilename.TcPOU, F_FILE_SplitPath.TcPOU, F_FILE_TIME_GT.TcPOU, F_FILE_ULargeToFileTime.TcPOU
//   POUs/METS/Common LIB/08_SOFTWARE LIB/IP Address FBs/ F_IP_AddressPort.TcPOU
//   POUs/METS/Common LIB/08_SOFTWARE LIB/Logger FBs/ FB_LOG_FileWriteError.TcPOU, FB_LOG_Handler.TcPOU
//   POUs/METS/Common LIB/08_SOFTWARE LIB/Maths FBs/ FB_CumulativeAverage.TcPOU, FB_Interval.TcPOU, FB_MovingAverage.TcPOU, FB_MovingAverageEvent.TcPOU, FB_MovingAverageTimer.TcPOU, FB_MovingWindowEvent.TcPOU, FB_MovingWindowTimer.TcPOU, F_ApplyTimeOffset.TcPOU, F_CompareSign.TcPOU, F_FileTimeToULarge.TcPOU, F_GetSign.TcPOU, F_Interpolate.TcPOU, F_ModuloPos.TcPOU, F_SafeDIV.TcPOU, F_ULargeToFileTime.TcPOU
//   POUs/METS/Common LIB/08_SOFTWARE LIB/Memory FBs/ FB_StructureMonitor.TcPOU, F_8BitsToByte.TcPOU, F_Checksum_CRC16.TcPOU, F_FiltredSetBitState16.TcPOU (not stored), F_GetBitState.TcPOU, F_PointerToByteADD.TcPOU, F_PointerToWordADD.TcPOU, F_SafeTo_UDINT.TcPOU, F_SetBitState.TcPOU
//   POUs/METS/Common LIB/08_SOFTWARE LIB/String FBs/Concat Function/ F_CONCAT3.TcPOU (not stored), F_CONCAT4.TcPOU (not stored), F_CONCAT5.TcPOU (not stored), F_CONCAT6.TcPOU (not stored), F_CONCAT7.TcPOU (not stored), F_CONCAT8.TcPOU (not stored), F_CONCAT9.TcPOU (not stored)
//   POUs/METS/Common LIB/08_SOFTWARE LIB/String FBs/ FB_ExtractAnyString.TcPOU, FB_ExtractLongString.TcPOU, FB_ExtractString.TcPOU, FB_ExtractString_v2.TcPOU (excluded from build), F_AddPadding.TcPOU, F_AddPaddingUDINT.TcPOU, F_CodeToHex.TcPOU, F_InvalidateASCIIChar.TcPOU, F_InvalidNumericChar.TcPOU, F_IsNumber.TcPOU, F_ReplaceLongSingleChar.TcPOU, F_ReplaceSingleChar.TcPOU, F_ReplaceLongSingleChar.TcPOU, F_StringAddPrefix.TcPOU, F_StringAddSuffix.TcPOU, F_StringWildcard.TcPOU (not stored), F_ValidateString.TcPOU, F_ValidateString_Code.TcPOU, F_WriteEscapeCharacters.TcPOU, F_ZeroPadString.TcPOU
//   POUs/METS/Common LIB/08_SOFTWARE LIB/String FBs/LongConcat Function/ F_LongCONCAT.TcPOU (not stored) (excluded from build), F_LongDELETE.TcPOU (not stored) (excluded from build), F_LongFIND.TcPOU (not stored) (excluded from build), F_LongLEFT.TcPOU (not stored) (excluded from build), F_LongMID.TcPOU (not stored) (excluded from build), F_LongRIGHT.TcPOU (not stored) (excluded from build), F_LongToLowCase.TcPOU (not stored) (excluded from build)
//   POUs/METS/Common LIB/08_SOFTWARE LIB/TcChecks/ CheckBounds.TcPOU (not stored) (excluded from build), CheckDivReal.TcPOU (not stored) (excluded from build), CheckRangeSigned.TcPOU (not stored), CheckRangeUnsigned.TcPOU (not stored)
//   POUs/METS/Common LIB/08_SOFTWARE LIB/TCP FBs/ FB_TCP_ClientPortCtrl.TcPOU, FB_TCP_ClientPortCtrl_V2.TcPOU (not stored), FB_TCP_CloseAllPorts.TcPOU (not stored), FB_TCP_ReceiveData_V2.TcPOU (not stored), FB_TCP_ReceiveLongString.TcPOU (not stored), FB_TCP_ReceiveString.TcPOU (not stored), FB_TCP_SendData.TcPOU (not stored), FB_TCP_ServerPortCtrl.TcPOU (not stored)
//   POUs/METS/Common LIB/08_SOFTWARE LIB/Timer FBs/ FB_Blink.TcPOU (not stored), FB_Debounce.TcPOU (not stored), FB_EventRate.TcPOU (not stored), FB_EventsPerHour.TcPOU (not stored), FB_LongShortPress.TcPOU (not stored), FB_Puls.TcPOU (not stored), FB_PulseGenerator.TcPOU (not stored), FB_PulseGenerator_Sync.TcPOU (not stored), FB_PulseTrain.TcPOU (not stored), FB_SignalDelay.TcPOU (not stored), FB_Slew.TcPOU (not stored), FB_SquareWave.TcPOU (not stored), FB_SquareWave_Sync.TcPOU (not stored), FB_StopWatch.TcPOU (not stored), FB_StopWatch_LREAL.TcPOU (not stored), FB_TaskTime.TcPOU (not stored) (excluded from build), FB_TimeDistance.TcPOU (not stored), FB_TOFR.TcPOU (not stored), FB_TONR.TcPOU (not stored), P_Puls.TcPOU (not stored)
//   POUs/METS/Common LIB/09_SYSTEM LIB/ClearQueue/ FB_SYSTEM_ClearCameraStatus.TcPOU (not stored), FB_SYSTEM_ClearCaseDataArray.TcPOU (not stored), FB_SYSTEM_ClearCasePackerArray.TcPOU (not stored), FB_SYSTEM_ClearHMIQueue.TcPOU (not stored), FB_SYSTEM_ClearMasterListArray.TcPOU (not stored), FB_SYSTEM_ClearOuterArray.TcPOU (not stored), FB_SYSTEM_ClearPackArray.TcPOU (not stored)
//   POUs/METS/Common LIB/09_SYSTEM LIB/PCM FB%27s/ FB_PCM_ReadFile.TcPOU (not stored), FB_PCM_SetData.TcPOU (not stored), FB_PCM_TrackingModeDecode.TcPOU (not stored), FB_PCM_Validate.TcPOU (not stored), FB_PCM_WriteFile.TcPOU (not stored)
//   POUs/METS/Common LIB/09_SYSTEM LIB/System Function/ F_SYSTEM_BoolToBArcodeType.TcPOU (not stored), F_SYSTEM_CameraMonitor.TcPOU (not stored), F_SYSTEM_DriverMonitor.TcPOU (not stored)
//   POUs/METS/Common LIB/09_SYSTEM LIB/System Time Function/ F_SYSTEM_ApplyTimeOffset.TcPOU (not stored), F_SYSTEM_Date.TcPOU (not stored), F_SYSTEM_DateCodeToDate.TcPOU (not stored), F_SYSTEM_DateCompare.TcPOU (not stored), F_SYSTEM_DateToDateCode.TcPOU (not stored), F_SYSTEM_DayOfYear.TcPOU (not stored), F_SYSTEM_DaysIntToTime.TcPOU (not stored), F_SYSTEM_HMIDateTime.TcPOU (not stored), F_SYSTEM_HMIDateTime_V2.TcPOU (not stored), F_SYSTEM_StringToTime.TcPOU (not stored), F_SYSTEM_SystemTimeAsISO8601.TcPOU (not stored), F_SYSTEM_SystemTimeOffsetToHHMM.TcPOU (not stored), F_SYSTEM_SystemTimeToCHM_Header.TcPOU (not stored), F_SYSTEM_SystemTimeToFolderName.TcPOU (not stored), F_SYSTEM_SystemTimeToOHMFolderName.TcPOU (not stored), F_SYSTEM_Time.TcPOU (not stored), F_SYSTEM_TimeFine.TcPOU (not stored), F_SYSTEM_TimeSuperFine.TcPOU (not stored), F_SYSTEM_ValidProduceDate.TcPOU (not stored)
//   POUs/METS/Common LIB/10_SIMULATOR LIB/Code Generator/ C91_FB_CharacterGenerator.TcPOU (not stored), C91_FB_OuterCodeAggregator.TcPOU (not stored), C91_FB_OuterCodeGenerator.TcPOU (not stored), C91_FB_PackCodeAggregator.TcPOU (not stored), C91_FB_PackCodeGenerator.TcPOU (not stored)
//   POUs/METS/Common LIB/10_SIMULATOR LIB/Code Generator/Code Generator/FB - Not used/ FB_CODE_BATSerializator.TcPOU (not stored)
//   POUs/METS/Common LIB/10_SIMULATOR LIB/Code Generator/Code Generator/ FB_CODE_CaseCodeGenerator.TcPOU (not stored), FB_CODE_OuterCodeGenerator.TcPOU (not stored), F_CODE_BATSerializator.TcPOU (not stored)
//   POUs/METS/Common LIB/10_SIMULATOR LIB/Code Generator/OLD/ C90_FB_CaseCodeGenerator.TcPOU (not stored) (excluded from build), C90_FB_CharacterGenerator.TcPOU (not stored) (excluded from build), C90_FB_Codes_Aggregator.TcPOU (not stored) (excluded from build), C90_FB_PackCodeGenerator.TcPOU (not stored) (excluded from build), C90_Generator.TcPOU (not stored) (excluded from build)
//   POUs/METS/METS General/00 Fast Task %28Devices%29/Automation Mode/CML SEQUENCE/ PRG_CML_01_InfeedCtrl.TcPOU (not stored), PRG_CML_02_LoweratorCtrl.TcPOU (not stored), PRG_CML_03_AdditionalConvCtrl.TcPOU (not stored) (excluded from build)
//   POUs/METS/METS General/00 Fast Task %28Devices%29/Automation Mode/LARS SEQUENCE/ PRG_LARS_01_TransportConvCtrl.TcPOU (not stored), PRG_LARS_02_GateSeparationCtrl.TcPOU (not stored), PRG_LARS_03_AddtitionalConvCtrl.TcPOU (not stored)
//   POUs/METS/METS General/00 Fast Task %28Devices%29/Automation Mode/SFLX SEQUENCE/ PRG_SFLX_01_TransportConvCtrl.TcPOU (not stored), PRG_SFLX_02_OutfeedConvCtrl.TcPOU (not stored), PRG_SFLX_03_AddtitionalConvCtrl.TcPOU (not stored)
//   POUs/METS/METS General/00 Fast Task %28Devices%29/ F00_Safety_Signals.TcPOU (not stored), F01_METS_SingleInputs.TcPOU (not stored), F02_METS_DoubleInputs.TcPOU (not stored), F04_PackAggrergationCtrl.TcPOU (not stored), F06_OuterAutomationCtrl.TcPOU (not stored), F08_OuterAggregationCtrl.TcPOU (not stored), F10_CasePackerDoorCtrl.TcPOU (not stored), F11_InfeedConvQueueCtrl.TcPOU (not stored), F11_InfeedConvQueueCtrl_V3.TcPOU (not stored) (excluded from build), F12_PackerQueuesCtrl.TcPOU (not stored), F13_CaseContentValidation.TcPOU (not stored), F14_CaseQueueControl.TcPOU (not stored), F15_CaseControlCACData.TcPOU (not stored), F18_ClearSystemQueues.TcPOU (not stored), F19_ClearInspectionStatistic.TcPOU (not stored), F20_HandScanner.TcPOU (not stored), F21_ContentHandScanner.TcPOU (not stored), F22_AggregationHandScanner.TcPOU (not stored), F25_CylindersCtrl.TcPOU (not stored), F26_EncodersCtrl.TcPOU (not stored), F30_PrintersCommCtrl.TcPOU (not stored), F32_InterimPrinter.TcPOU (not stored), F33_OuterPrinters.TcPOU (not stored), F33_OuterPrinters_v2_Evo.TcPOU (not stored) (excluded from build), F34_CasePrinter.TcPOU (not stored), F40_StationManager.TcPOU (not stored), F45_EventLoggerExt.TcPOU (not stored), F60_METS_Outputs.TcPOU (not stored), F95_CameraTest.TcPOU (not stored), F96_CHMTester.TcPOU (not stored) (excluded from build), F97_CodesGenerator.TcPOU (not stored) (excluded from build), F98_TCPServer.TcPOU (not stored) (excluded from build), F99_DiagnosticBlock.TcPOU (not stored)
//   POUs/METS/METS General/00 Fast Task %28Devices%29/Outer Aggregation Mode/CML/ PRG_CML_SynchroAggregation.TcPOU (not stored), PRG_CML_ValidationAsConfirmation.TcPOU (not stored)
//   POUs/METS/METS General/00 Fast Task %28Devices%29/Outer Aggregation Mode/LARS/ PRG_LARS_SynchroAggregation.TcPOU (not stored), PRG_LARS_ValidationAsConfirmation.TcPOU (not stored)
//   POUs/METS/METS General/00 Fast Task %28Devices%29/Outer Aggregation Mode/SFLX/ PRG_SFLX_NoValidationCamera.TcPOU (not stored), PRG_SFLX_ValidationAsConfirmation.TcPOU (not stored)
//   POUs/METS/METS General/00 Fast Task %28Devices%29/Pack Aggregation Mode/PAOL SEQUENCE/2CAM_METSONE/ PRG_PAOL_01_LightboxScanersCtrl.TcPOU (not stored)
//   POUs/METS/METS General/00 Fast Task %28Devices%29/Pack Aggregation Mode/PAOL SEQUENCE/3CAM_LIGHTBOX/ PRG_PAOL_02_LightboxScanersCtrl.TcPOU (not stored), PRG_PAOL_03_LightboxSeparatorCtrl.TcPOU (not stored)
//   POUs/METS/METS General/00 Fast Task %28Devices%29/Pack Aggregation Mode/PLAS SEQUENCE/T01_CW_GD/ PRG_PLAS_01_PrimaryMasterListCtrl.TcPOU (not stored), PRG_PLAS_02_PackAggregationCtrl.TcPOU (not stored), PRG_PLAS_03_PackToStackerCtrl.TcPOU (not stored), PRG_PLAS_04_CompleteOuterCtrl.TcPOU (not stored)
//   POUs/METS/METS General/00 Fast Task %28Devices%29/Pack Aggregation Mode/PLAS SEQUENCE/T02_NCW_GD/ PRG_PLAS_05_PrimaryMasterListCtrl.TcPOU (not stored), PRG_PLAS_06_PackAggregationCtrl.TcPOU (not stored), PRG_PLAS_07_PackToStackerCtrl.TcPOU (not stored), PRG_PLAS_08_InterimCamCtrl.TcPOU (not stored), PRG_PLAS_09_CompleteOuterCtrl.TcPOU (not stored)
//   POUs/METS/METS General/00 Fast Task %28Devices%29/Pack Aggregation Mode/PLAS SEQUENCE/T03_NCW_FOCKE/ PRG_PLAS_10_PrimaryMasterListCtrl.TcPOU (not stored), PRG_PLAS_11_PackAggregationCtrl.TcPOU (not stored), PRG_PLAS_12_MovePacksToOCVCtrl.TcPOU (not stored), PRG_PLAS_13_InterimCamCtrl.TcPOU (not stored), PRG_PLAS_14_CompleteOuterCtrl.TcPOU (not stored)
//   POUs/METS/METS General/00 Fast Task %28Devices%29/Pack Aggregation Mode/PLAS SEQUENCE/T04_NCW_FOCKE_HYBRID/ PRG_PLAS_15_PrimaryMasterListCtrl.TcPOU (not stored), PRG_PLAS_16_PackAggregationCtrl.TcPOU (not stored), PRG_PLAS_17_MovePacksToOCVCtrl.TcPOU (not stored), PRG_PLAS_18_InterimCamCtrl.TcPOU (not stored), PRG_PLAS_19_CompleteOuterCtrl.TcPOU (not stored), PRG_PLAS_20_LightboxSeparatorCtrl.TcPOU (not stored)
//   POUs/METS/METS General/03 xFast Task %28Data Base%29/ X00_TimeLogger.TcPOU (not stored) (excluded from build), X02_Database.TcPOU (not stored) (excluded from build), X03_CyclicReport.TcPOU (not stored) (excluded from build), X10_xFastOutputs.TcPOU (not stored) (excluded from build)
//   POUs/METS/ T00_FAST.TcPOU, T01_CONTROL.TcPOU, T02_ACCESSORY.TcPOU, T03_xFAST.TcPOU
//   POUs/TcUnit/FB_ExtractAnyStringTests/ FB_ExtractAnyStringTests.TcPOU, PRG_ExtractAnyStringManual.TcPOU
//   POUs/TcUnit/FB_ExtractStringTests/ FB_ExtratcStringTests.TcPOU, PRG_ExtractStringManual.TcPOU
//   POUs/TcUnit/FB_LOGHandlerTests/ FB_LogHandlerTests.TcPOU, PRG_LogHandlerManual.TcPOU
//   POUs/TcUnit/FUN_ReplaceLongSingleCharTests/ FB_ReplaceLongStringCharTests.TcPOU, PRG_ReplaceLongSingleCharManual.TcPOU
//   POUs/TcUnit/ PRG_TEST.TcPOU
//   POUs/_Exclude/DUT/ E_LOG_HandlerName_OLD.TcDUT (excluded from build), ST_SYSTEM_Config_old.TcDUT (excluded from build)
//   POUs/_Exclude/FSS2/ FB_FSS2_BuildXMLData.TcPOU (excluded from build), FB_FSS2_BuildXMLDataForGMES.TcPOU (excluded from build), FB_FSS2_WriteFile.TcPOU (excluded from build), FB_FSS2_WriteFileForGMES.TcPOU (excluded from build), FB_FSS2_XMLImageGenerator.TcPOU (excluded from build)
//   POUs/_Exclude/OAC FBs/ FB_OAC_BuildXMLData.TcPOU (excluded from build), FB_OAC_ClearArchive.TcPOU (excluded from build), FB_OAC_FindFile.TcPOU (excluded from build), FB_OAC_WriteFile.TcPOU (excluded from build)
//   POUs/_Exclude/OCV FBs/ FB_OCV_BuildXMLData.TcPOU (excluded from build), FB_OCV_ClearArchive.TcPOU (excluded from build), FB_OCV_FindFile.TcPOU (excluded from build), FB_OCV_FindFileWithError.TcPOU (excluded from build), FB_OCV_WriteFile.TcPOU (excluded from build)
//   POUs/_Exclude/v1/ FB_CAC_MoveToArchive.TcPOU (excluded from build), FB_CAC_PopulateMinimalOuterData.TcPOU (excluded from build), FB_CAC_WriteFile.TcPOU (excluded from build)
//   POUs/_Exclude/v1_1/ FB_CHM_BiuldXMLImige.TcPOU (excluded from build), FB_CHM_XMLImageGenerator.TcPOU (excluded from build)
//   POUs/_Exclude/v2/ FB_CAC_MoveFromArchive.TcPOU (excluded from build), FB_CAC_RestoreOAC.TcPOU (excluded from build), FB_CAC_WriteFile_v2.TcPOU (excluded from build), FB_CAC_WriteToArchive_v2.TcPOU (excluded from build)
//   POUs/_Exclude/v2_1/ FB_CHM_BiuldXMLImige_v2.TcPOU (excluded from build), FB_CHM_HierachyGenerator.TcPOU (excluded from build)
//   POUs/_Exclude/v3/ FB_CHM_BiuldXMLImige_v3.TcPOU (excluded from build)
//   POUs/_Exclude/XML/ FB_CX_NVData_XMLFile_32K.TcPOU (excluded from build), FB_CX_NVData_XMLFile_4K.TcPOU (excluded from build)

CONFIGURATION PLC_Convert
    RESOURCE PLC ON TwinCAT3
        TASK Control_Task(INTERVAL := T#12ms, PRIORITY := 22);
        TASK xFast_Task(INTERVAL := T#1ms, PRIORITY := 20);
        TASK Fast_Task(INTERVAL := T#3ms, PRIORITY := 21);
        TASK Accessory_Task(INTERVAL := T#100000us, PRIORITY := 23);
        TASK TcUnit_Task(INTERVAL := T#10ms, PRIORITY := 25);
        PROGRAM T01_CONTROL WITH Control_Task : T01_CONTROL;
        PROGRAM T03_xFAST WITH xFast_Task : T03_xFAST;
        PROGRAM T00_FAST WITH Fast_Task : T00_FAST;
        PROGRAM T02_ACCESSORY WITH Accessory_Task : T02_ACCESSORY;
        PROGRAM PRG_TEST WITH TcUnit_Task : PRG_TEST;
    END_RESOURCE
END_CONFIGURATION

// ---- Data types/METS/ADS Symobol/E_SYMBOL_AccessState.TcDUT
TYPE E_SYMBOL_AccessState :
(
	E_SYMBOL_IDLE,
	E_SYMBOL_GETSYMBOLINFO,
	E_SYMBOL_READDATA,
	E_SYMBOL_WRITEDATA,
	E_SYMBOL_DONE
);
END_TYPE

// ---- Data types/METS/ADS Symobol/E_SYMBOL_AdsStates.TcDUT
TYPE E_SYMBOL_AdsStates :
(
	ADSSTATES_INVALID :=0,
	ADSSTATES_IDLE :=1,
	ADSSTATES_RESET :=2,
	ADSSTATES_INIT :=3,
	ADSSTATES_START :=4,
	ADSSTATES_RUN :=5,
	ADSSTATES_STOP :=6,
	ADSSTATES_SAVECFG :=7,
	ADSSTATES_LOADCFG :=8,
	ADSSTATES_POWERFAILURE :=9,
	ADSSTATES_POWERGOOD :=10,
	ADSSTATES_ERROR :=11
);
END_TYPE

// ---- Data types/METS/ADS Symobol/ST_SYMBOL_AddressInfo.TcDUT
TYPE ST_SYMBOL_AddressInfo :	(* 8 bytes *)
STRUCT
	pSymAddr	: 	DWORD;
	nSymSize	:	UDINT;
END_STRUCT
END_TYPE

// ---- Data types/METS/AI Codes And Validation/E_CodeAIType.TcDUT
TYPE E_CodeAIType :
STRUCT
	GTIN 			: 	INT := 1;
	BatchID 			: 	INT := 10;
	SerialCode		: 	INT := 21;
	ProductionOrder 	: 	INT := 91;
	CryptoCode		: 	INT := 93;
	RSKU 			: 	INT := 240;
	MRP				:	INT := 8005;
	BrandSpecification 	:	INT := 92;
	ProduceDate		:	INT := 94;
	UserField3		:	INT;
END_STRUCT
END_TYPE

// ---- Data types/METS/AI Codes And Validation/E_CodeType.TcDUT
TYPE E_CodeType :
(
	E_NONE,
	E_PACK,
	E_INTERIM,
	E_OUTER,
	E_CASE

);
END_TYPE

// ---- Data types/METS/AI Codes And Validation/GS1_Standard/E_GS1_CodeAIType.TcDUT
TYPE E_GS1_CodeAIType :
(
	GS1_00		:= 0,		(*GS1 Not defined*)
	GS1_01		 :=1,		(***********Global Trade Item Number (GTIN)	N2+N14*************)
	GS1_10		:=10,		(***********Batch or lot number	N2+X..20*************)
	GS1_11		:=11,		(***********Production date (YYMMDD)		N2+N6*************)
	GS1_15		:=15,		(***********Best before date (YYMMDD)			N2+N6*************)
	GS1_17		:=17,		(***********Expiration date (YYMMDD)		N2+N6*************)
	GS1_21		:=21,		(***********Serial number		N2+X..20*************)
	GS1_240		:=240,	(***********Additional product identification assigned by the manufacturer	N3+X..30*************)
	GS1_8005		:=8005,	(***********Price per unit of measure	N4+N6*************)
	GS1_8006		:=8006,	(***********Identification of an individual trade item piece	N4+N14+N2+N2*************)
	GS1_8008		:=8008,	(***********Date and time of production		N4+N8+N..4*************)
	GS1_91		:=91,		(***********Company internal information	N2+X..90*************)
	GS1_92		:=92,		(***********Company internal information	N2+X..90*************)
	GS1_93		:=93,		(***********Company internal information	N2+X..90*************)
	GS1_94		:=94,		(***********Company internal information	N2+X..90*************)
	NON_GS1_01		:=10001,	(***********Non GS1 - user defined		X..255*************)
	NON_GS1_02		:=10002,	(***********Non GS1 - user defined		X..255*************)
	NON_GS1_03		:=10003,	(***********Non GS1 - user defined		X..255*************)
	NON_GS1_04		:=10004,	(***********Non GS1 - user defined		X..255*************)
	NON_GS1_05		:=10005,	(***********Non GS1 - user defined		X..255*************)
	NON_GS1_06		:=10006,	(***********Non GS1 - user defined		X..255*************)
	NON_GS1_07		:=10007,	(***********Non GS1 - user defined		X..255*************)
	NON_GS1_08		:=10008,	(***********Non GS1 - user defined		X..255*************)
	NON_GS1_09		:=10009,	(***********Non GS1 - user defined		X..255*************)
	NON_GS1_10		:=10010	(***********Non GS1 - user defined		X..255*************)
);
END_TYPE

// ---- Data types/METS/AI Codes And Validation/GS1_Standard/E_GS1_CodeLvl.TcDUT
TYPE E_GS1_CodeLvl :
(
	E_LVL_NONE,
	E_LEVEL1,
	E_LEVEL2,
	E_LEVEL3
);
END_TYPE

// ---- Data types/METS/AI Codes And Validation/GS1_Standard/ST_GS1_AI_Attributs.TcDUT
TYPE ST_GS1_AI_Attributs :
STRUCT
	sDataField 	: T_MaxString;
	bDataChanged	: BOOL;
	sAI_Id		: STRING(5);
	eGS1_AI		: E_GS1_CodeAIType;
	bFixed		: BOOL;
	nLength		: UINT;
END_STRUCT
END_TYPE

// ---- Data types/METS/AI Codes And Validation/GS1_Standard/ST_GS1_AI_Definition.TcDUT
TYPE ST_GS1_AI_Definition :
STRUCT
	sDotCode_CI	: STRING(3) := ']j';			(* GS1 marker (FNC1 Carrier Identifiers for DataMatrix barcode *)
	sDMC_CI		: STRING(3) := ']d2';			(* GS1 marker (FNC1 Carrier Identifiers for DataMatrix barcode *)
	sCode128_CI	: STRING(3) := ']c1';			(* GS1 marker (FNC1 Carrier Identifiers for Code128 barcode *)
	stAI_01_Lvl1	: ST_GS1_AI_Attributs := (sAI_Id:='01', eGS1_AI:=GS1_01, bFixed:= TRUE, nLength:=14);	(***********N2+N14*************)
	stAI_01_Lvl2	: ST_GS1_AI_Attributs := (sAI_Id:='01', eGS1_AI:=GS1_01, bFixed:= TRUE, nLength:=14);	(***********N2+N14*************)
	stAI_01_Lvl3	: ST_GS1_AI_Attributs := (sAI_Id:='01', eGS1_AI:=GS1_01, bFixed:= TRUE, nLength:=14);	(***********N2+N14*************)
	stAI_10		: ST_GS1_AI_Attributs := (sAI_Id:='10', eGS1_AI:=GS1_10, bFixed:= FALSE, nLength:=20);	(***********N2+X..20*************)
	stAI_11		: ST_GS1_AI_Attributs := (sAI_Id:='11', eGS1_AI:=GS1_11, bFixed:= TRUE, nLength:=6);	(***********N2+N6*************)
	stAI_15		: ST_GS1_AI_Attributs := (sAI_Id:='15', eGS1_AI:=GS1_15, bFixed:= TRUE, nLength:=6);	(***********N2+N6*************)
	stAI_17		: ST_GS1_AI_Attributs := (sAI_Id:='17', eGS1_AI:=GS1_17, bFixed:= TRUE, nLength:=6);	(***********N2+N6*************)
	stAI_21		: ST_GS1_AI_Attributs := (sAI_Id:='21', eGS1_AI:=GS1_21, bFixed:= FALSE, nLength:=20);	(***********N2+X..20*************)
	stAI_240		: ST_GS1_AI_Attributs := (sAI_Id:='240', eGS1_AI:=GS1_240, bFixed:= FALSE, nLength:=30);		(***********N3+X..30*************)
	stAI_8005		: ST_GS1_AI_Attributs := (sAI_Id:='8005', eGS1_AI:=GS1_8005, bFixed:= TRUE, nLength:=6);		(***********N4+N6*************)
	stAI_8006		: ST_GS1_AI_Attributs := (sAI_Id:='8006', eGS1_AI:=GS1_8006, bFixed:= TRUE, nLength:=18);	(***********N4+N14+N2+N2*************)
	stAI_8008		: ST_GS1_AI_Attributs := (sAI_Id:='8008', eGS1_AI:=GS1_8008, bFixed:= TRUE, nLength:=12);	(***********N4+N8+N..4*************)
	stAI_91		: ST_GS1_AI_Attributs := (sAI_Id:='91', eGS1_AI:=GS1_91, bFixed:= FALSE, nLength:=90);		(***********N2+X..90*************)
	stAI_92		: ST_GS1_AI_Attributs := (sAI_Id:='92', eGS1_AI:=GS1_92, bFixed:= FALSE, nLength:=90);		(***********N2+X..90*************)
	stAI_93		: ST_GS1_AI_Attributs := (sAI_Id:='93', eGS1_AI:=GS1_93, bFixed:= FALSE, nLength:=90);		(***********N2+X..90*************)
	stAI_94		: ST_GS1_AI_Attributs := (sAI_Id:='94', eGS1_AI:=GS1_94, bFixed:= FALSE, nLength:=90);		(***********N2+X..90*************)

	stNON_GS1_01		: ST_GS1_AI_Attributs := (sAI_Id:='10001', eGS1_AI:=NON_GS1_01, bFixed:= FALSE, nLength:=255);		(***********X..255*************)
	stNON_GS1_02		: ST_GS1_AI_Attributs := (sAI_Id:='10002', eGS1_AI:=NON_GS1_02, bFixed:= FALSE, nLength:=255);		(***********X..255*************)
	stNON_GS1_03		: ST_GS1_AI_Attributs := (sAI_Id:='10003', eGS1_AI:=NON_GS1_03, bFixed:= FALSE, nLength:=255);		(***********X..255*************)
	stNON_GS1_04		: ST_GS1_AI_Attributs := (sAI_Id:='10004', eGS1_AI:=NON_GS1_04, bFixed:= FALSE, nLength:=255);		(***********X..255*************)
	stNON_GS1_05		: ST_GS1_AI_Attributs := (sAI_Id:='10005', eGS1_AI:=NON_GS1_05, bFixed:= FALSE, nLength:=255);		(***********X..255*************)
	stNON_GS1_06		: ST_GS1_AI_Attributs := (sAI_Id:='10006', eGS1_AI:=NON_GS1_06, bFixed:= FALSE, nLength:=255);		(***********X..255*************)
	stNON_GS1_07		: ST_GS1_AI_Attributs := (sAI_Id:='10007', eGS1_AI:=NON_GS1_07, bFixed:= FALSE, nLength:=255);		(***********X..255*************)
	stNON_GS1_08		: ST_GS1_AI_Attributs := (sAI_Id:='10008', eGS1_AI:=NON_GS1_08, bFixed:= FALSE, nLength:=255);		(***********X..255*************)
	stNON_GS1_09		: ST_GS1_AI_Attributs := (sAI_Id:='10009', eGS1_AI:=NON_GS1_09, bFixed:= FALSE, nLength:=255);		(***********X..255*************)
	stNON_GS1_10		: ST_GS1_AI_Attributs := (sAI_Id:='10010', eGS1_AI:=NON_GS1_10, bFixed:= FALSE, nLength:=255);		(***********X..255*************)

END_STRUCT
END_TYPE

// ---- Data types/METS/AI Codes And Validation/GS1_Standard/ST_GS1_CodeInfo.TcDUT
TYPE ST_GS1_CodeInfo :
STRUCT
	eCodeLvlType					:	E_GS1_CodeLvl;

	nMinLength					: 	INT;
	nEntireLength					:	INT;
	bValidateEntireLength			: 	BOOL;
	nNumberOfAIs					:	INT;

	stGS1_Field 					: ARRAY[1..cMAX_VALIDATION_ITEMS] OF 	ST_GS1_CodeValidation	;

	(*stGS1_Field01 				:	ST_GS1_CodeValidation	;
	stGS1_Field02 					:	ST_GS1_CodeValidation	;
	stGS1_Field03 					:	ST_GS1_CodeValidation	;
	stGS1_Field04 					:	ST_GS1_CodeValidation	;
	stGS1_Field05					:	ST_GS1_CodeValidation	;
	stGS1_Field06					:	ST_GS1_CodeValidation	;
	stGS1_Field07		 			:	ST_GS1_CodeValidation	;
	stGS1_Field08					:	ST_GS1_CodeValidation	;
	stGS1_Field09					:	ST_GS1_CodeValidation	;
	stGS1_Field10					:	ST_GS1_CodeValidation	;*)

END_STRUCT
END_TYPE

// ---- Data types/METS/AI Codes And Validation/GS1_Standard/ST_GS1_CodeValidation.TcDUT
TYPE ST_GS1_CodeValidation :
STRUCT

	bValidate 			:	BOOL;
	sFieldName		:	STRING(15)	:='';

	sStartAI 			: 	STRING(6)		:= '';
	sEndAI 			: 	STRING(6) 	:= '';
	nCodeStartPos		:	INT;
	nCodeLength		:	INT;

	eGS1_AIType		: 	E_GS1_CodeAIType 	:= GS1_00;

(* If sStartAI is empty, then use nCodeStartPos, else find sStartAI in code for start position *)
(* If sEndAI is empty then use nCodeLength, else find sEndAI in code for end position*)

(*General Application Idendifiers (AI) Description:
	01:		GTIN
	10: 		Batch ID/WorkOrderID
	21: 		Serial Code
	91:		Production Order/WorkCenterID
	93:		Crypto
	240:		RSKU
*)

END_STRUCT
END_TYPE

// ---- Data types/METS/AI Codes And Validation/GS1_Standard/ST_GS1_Decode_AI.TcDUT
TYPE ST_GS1_Decode_AI :
STRUCT
	sAI_Id		: STRING(5);
	bFixed		: BOOL;
	nLength		: UINT;
END_STRUCT
END_TYPE

// ---- Data types/METS/AI Codes And Validation/ST_CodeInfo.TcDUT
TYPE ST_CodeInfo :
STRUCT
	eCodeType					:	E_CodeType;

	nMinLength					: 	INT;
	nEntireLength					:	INT;
	bValidateEntireLength			: 	BOOL;
	nNumberOfAIs					:	INT;

	stGTIN 						:	ST_CodeValidation	:=		(sFieldName :='GTIN',						bNameEditable := FALSE, 		nGS1_AI := 1);
	stBatchID 						:	ST_CodeValidation	:=		(sFieldName :='BatchID', 				bNameEditable := FALSE, 		nGS1_AI := 10);
	stSerialCode 					:	ST_CodeValidation	:=		(sFieldName :='SerialCode', 			bNameEditable := FALSE, 		nGS1_AI := 21);
	stProductionOrder 				:	ST_CodeValidation	:=		(sFieldName :='ProductionOrder', 		bNameEditable := FALSE, 		nGS1_AI := 91);
	stCryptoCode					:	ST_CodeValidation	:=		(sFieldName :='CryptoCode', 			bNameEditable := FALSE, 		nGS1_AI := 93);
	stRSKU						:	ST_CodeValidation	:=		(sFieldName :='RSKU', 						bNameEditable := FALSE, 		nGS1_AI := 240);
	stMRP		 				:	ST_CodeValidation	:=		(sFieldName :='MRP', 						bNameEditable := FALSE, 		nGS1_AI := 8005);
	stBrandSpecification			:	ST_CodeValidation	:=		(sFieldName :='BrandSpec',			bNameEditable := FALSE, 		nGS1_AI := 92);
	stProduceDate					:	ST_CodeValidation	:=		(sFieldName :='ProduceDate',			bNameEditable := TRUE, 		nGS1_AI := 94);
	stUserField3					:	ST_CodeValidation	:=		(sFieldName :='',						bNameEditable := TRUE, 		nGS1_AI := 95);

END_STRUCT
END_TYPE

// ---- Data types/METS/AI Codes And Validation/ST_CodeValidation.TcDUT
TYPE ST_CodeValidation :
STRUCT
	bValidate 			:	BOOL;

	sFieldName		:	STRING(15)	:='';
	bNameEditable	:	BOOL;
	nListPosition		: 	BYTE;

	sStartAI 			: 	STRING(6)		:= '';
	sEndAI 			: 	STRING(6) 	:= '';
	nCodeStartPos		:	INT;
	nCodeLength		:	INT;

	nGS1_AI			: 	INT;

(* If sStartAI is empty, then use nCodeStartPos, else find sStartAI in code for start position *)
(* If sEndAI is empty then use nCodeLength, else find sEndAI in code for end position*)

(*General Application Idendifiers (AI) Description:
	01:		GTIN
	10: 		Batch ID
	21: 		Serial Code
	91:		Production Order
	93:		Crypto
	240:		RSKU
*)

END_STRUCT
END_TYPE

// ---- Data types/METS/AI Codes And Validation/ST_RejectItems.TcDUT
TYPE ST_RejectItems :
STRUCT
	nRejectID			: UINT;
	sMetsDisplayCode	: T_RejectCode; (*this is what is displayed on our HMI - nn is replaced by the number of failures/successes*)
	sMetsSearchCode	: STRING(50); (*this is what to search for when changing the reject reason for FSS*)
	sFssSendCode		: T_FSS_RejecCode; (*this is what to send to FSS*)
END_STRUCT
END_TYPE

// ---- Data types/METS/AI Codes And Validation/ST_RejectReasonsForCase.TcDUT
TYPE ST_RejectReasonsForCase :
STRUCT
	stValError:				ST_RejectItems :=(		nRejectID := 301,
														sMetsDisplayCode:='XXVALnnXX',
														sMetsSearchCode:='VAL',
														sFssSendCode:='Validation_DeferredOuter');

	stOACError:				ST_RejectItems :=(	nRejectID := 302,
														sMetsDisplayCode:='XXOACnnXX',
														sMetsSearchCode:='OAC',
														sFssSendCode:='Validation_DeferredPackData');

	stINVError:				ST_RejectItems :=(	nRejectID := 303,
														sMetsDisplayCode:='XXINVnnXX',
														sMetsSearchCode:='INV',
														sFssSendCode:='Validation_BelowAcceptanceLevel');

	stDUPError:				ST_RejectItems :=(	nRejectID := 304,
														sMetsDisplayCode:='XXDUPn1-n2XX',
														sMetsSearchCode:='DUP',
														sFssSendCode:='Validation_DuplicateData');

	stPackNotLinedError:		ST_RejectItems :=(	nRejectID := 305,
														sMetsDisplayCode:='XXPACKnnXX',
														sMetsSearchCode:='XPACK',
														sFssSendCode:='Validation_BadPackCode');

	stOuterGTINError:		ST_RejectItems :=(		nRejectID := 306,
														sMetsDisplayCode:='XXOUTERGTINnnXX',
														sMetsSearchCode:='OUTERGTIN',
														sFssSendCode:='Validation_BadOuterCode');

	stOuterSerialError:		ST_RejectItems :=(		nRejectID := 307,
														sMetsDisplayCode:='XXOUTERSERnnXX',
														sMetsSearchCode:='OUTERSER',
														sFssSendCode:='Validation_BadOuterCode');

	stOuterRSKUError:		ST_RejectItems :=(		nRejectID := 308,
														sMetsDisplayCode:='XXOUTERSKUnnXX',
														sMetsSearchCode:='OUTERSKU',
														sFssSendCode:='Validation_BadOuterCode');

	stNoCaseLabelError:		ST_RejectItems :=(		nRejectID := 309,
														sMetsDisplayCode:='XXNOCASELABELXX',
														sMetsSearchCode:='NOCASELABEL',
														sFssSendCode:='NoReadCase');

	stCasePackerReject:		ST_RejectItems :=(		nRejectID := 310,
														sMetsDisplayCode:='XXCASEPACKERREJECTXX',
														sMetsSearchCode:='CASEPACKERREJECT',
														sFssSendCode:='CasePackerReject');

	stDoorGuardReject:		ST_RejectItems :=(		nRejectID := 311,
														sMetsDisplayCode:='XXDOORGUARDREJECTXX',
														sMetsSearchCode:='DOORGUARDREJECT',
														sFssSendCode:='DoorReject');

	stCaseLabelGtinError:	ST_RejectItems :=(		nRejectID := 312,
														sMetsDisplayCode:='XXCASEGTINXX',
														sMetsSearchCode:='CASEGTIN',
														sFssSendCode:='Validation_BadLabel');

	stCaseLabelRskuError:	ST_RejectItems :=(		nRejectID := 313,
														sMetsDisplayCode:='XXCASESKUXX',
														sMetsSearchCode:='CASESKU',
														sFssSendCode:='Validation_BadLabel');

	stCaseLabelProductionOrderError:	ST_RejectItems :=(	nRejectID := 314,
														sMetsDisplayCode:='XXCASEPRODXX',
														sMetsSearchCode:='CASEPROD',
														sFssSendCode:='Validation_BadLabel');

	stCaseLabelBatchIDError:	ST_RejectItems :=(		nRejectID := 315,
														sMetsDisplayCode:='XXCASEBATCHXX',
														sMetsSearchCode:='CASEBATCH',
														sFssSendCode:='Validation_BadLabel');

	stCaseLabelSerialCodeError:	ST_RejectItems :=(	nRejectID := 316,
														sMetsDisplayCode:='XXCASESERIALCODEXX',
														sMetsSearchCode:='CASESERIALCODE',
														sFssSendCode:='Validation_BadLabel');

	stCaseLabelDuplicate:	ST_RejectItems :=(		nRejectID := 317,
														sMetsDisplayCode:='XXDUPCASELABELXX',
														sMetsSearchCode:='DUPCASELABEL',
														sFssSendCode:='Validation_CaseDuplicate');

	stCaseNoCaseData:	ST_RejectItems :=(			nRejectID := 318,
														sMetsDisplayCode:='XXNOCASEDATAXX',
														sMetsSearchCode:='NOCASEDATA',
														sFssSendCode:='Integrity_TooFewItemsCase');

	stCaseBarcodeInvalidLength:	ST_RejectItems :=(	nRejectID := 319,
														sMetsDisplayCode:='XXCASECODELENGTHXX',
														sMetsSearchCode:='CASECODELENGTH',
														sFssSendCode:='Validation_BadLabel');

	stCaseDBInvalidCheck	:	ST_RejectItems :=(	nRejectID := 320,
														sMetsDisplayCode:='XXCACDBINVALIDXX',
														sMetsSearchCode:='CACDBINVALID',
														sFssSendCode:='Validation_DBInvalid');

	stCaseWhitelistInvalidCheck	:	ST_RejectItems :=(	nRejectID := 321,
														sMetsDisplayCode:='XXOHMWHITELISTXX',
														sMetsSearchCode:='OHMWHITELIST',
														sFssSendCode:='Validation_OHMWhitelistInvalid');

	stOuterBrandError				:	ST_RejectItems :=(	nRejectID := 322,
														sMetsDisplayCode:='XXOUTERSBRANDnnXX',
														sMetsSearchCode:='OUTERSBRAND',
														sFssSendCode:='Validation_BadOuterCode');

	stCaseLabelBrandCodeError:	ST_RejectItems :=(	nRejectID := 323,
														sMetsDisplayCode:='XXCASEBRANDXX',
														sMetsSearchCode:='CASEBRAND',
														sFssSendCode:='Validation_BadLabel');

	stUnknownCaseReject:		ST_RejectItems :=(	nRejectID := 300,
														sMetsDisplayCode:='UnknownReason',
														sMetsSearchCode:='UnknownReason',
														sFssSendCode:='UnknownReason');

END_STRUCT
END_TYPE

// ---- Data types/METS/AI Codes And Validation/ST_RejectReasonsForOuter.TcDUT
TYPE ST_RejectReasonsForOuter :
STRUCT
	stOuterBarcodeGtinError:		ST_RejectItems :=(	nRejectID := 201,
															sMetsDisplayCode:='Outer code invalid GTIN',
															sMetsSearchCode:='GTIN',
															sFssSendCode:='WrongMasterData');

	stOuterBarcodeRskuError:	ST_RejectItems :=(	nRejectID := 202,
															sMetsDisplayCode:='Outer code invalid RSKU',
															sMetsSearchCode:='RSKU',
															sFssSendCode:='WrongMasterData');

	stOuterCodeSerialError:		ST_RejectItems :=(	nRejectID := 203,
															sMetsDisplayCode:='Outer code invalid lenght Serial Code',
															sMetsSearchCode:='Serial',
															sFssSendCode:='Validation_BadCode');

	stOuterBarcodeInvalidLength:	ST_RejectItems :=(	nRejectID := 204,
															sMetsDisplayCode:='Outer code invalid Length',
															sMetsSearchCode:='Length',
															sFssSendCode:='Validation_BadCode');

	stOuterBarcodeNotRead:		ST_RejectItems :=(	nRejectID := 205,
															sMetsDisplayCode:='Outer Label Code Not Read',
															sMetsSearchCode:='Outer Label Code Not Read',
															sFssSendCode:='NoReadOuter');

	stOuterBarcodeDuplicate:	ST_RejectItems :=(	nRejectID := 206,
															sMetsDisplayCode:='Outer code duplicate',
															sMetsSearchCode:='code duplicate',
															sFssSendCode:='Validation_OuterDup');

	stOuterDataNotFound:		ST_RejectItems :=(	nRejectID := 207,
															sMetsDisplayCode:='Outer data (OAC) not found',
															sMetsSearchCode:='(OAC) not found',
															sFssSendCode:='NoReadOuterData');

	stOuterGeneralCodeError:	ST_RejectItems :=(	nRejectID := 208,
															sMetsDisplayCode:='No Codes Read At Aggregation Station',
															sMetsSearchCode:='No Codes Read At Aggregation Station',
															sFssSendCode:='Validation_General');

	stOuterTimeOutValidation:	ST_RejectItems :=(	nRejectID := 209,
															sMetsDisplayCode:='Outer Validation Timeout',
															sMetsSearchCode:='Validation Timeout',
															sFssSendCode:='Validation_General');

(*Outer general erros related to pack codes only - barcode validation - OK*)

	stOuterDuplicatedPackCodesFound:		ST_RejectItems :=(	nRejectID := 210,
															sMetsDisplayCode:='Outer contain duplicate pack codes',
															sMetsSearchCode:='duplicate pack codes',
															sFssSendCode:='Validation_PackDup');

	stOuterPackCodeDataNotFound:		ST_RejectItems :=(	nRejectID := 211,
															sMetsDisplayCode:='Outer - Pack codes data (OCV) not found',
															sMetsSearchCode:='OCV',
															sFssSendCode:='NoPacksCodeData');

	stOuterConfirmCodeNotRead:			ST_RejectItems :=(	nRejectID := 212,
															sMetsDisplayCode:= 'Interim code(s) not read',
															sMetsSearchCode:='Interim code(s) not read',
															sFssSendCode:='NoPackCodeData');

	stOuterPackCodeNotRead:				ST_RejectItems :=(	nRejectID := 213,
															sMetsDisplayCode:= 'Outer acceptance level - n1 of n2 pack codes read',
															sMetsSearchCode:='acceptance level',
															sFssSendCode:='Tolerance_PackNoRead');

	stOuterPackCodeInvalid:				ST_RejectItems :=(	nRejectID := 214,
															sMetsDisplayCode:= 'Outer - invalid pack code(s) found',
															sMetsSearchCode:='Outer - invalid pack',
															sFssSendCode:='Tolerance_PackInv');

(*Outer external rejeqt for quality - barcode validation - OK, pack codes(s) validation - OK*)

	stOuterQAReject:			ST_RejectItems :=(	nRejectID := 215,
															sMetsDisplayCode:='Outer QA Reject',
															sMetsSearchCode:='QA',
															sFssSendCode:='QA_Reject');

	stOuterPackCodeDBError:				ST_RejectItems :=(	nRejectID := 216,
															sMetsDisplayCode:= 'Number Pack code not found - n1 of n2 - DB Error',
															sMetsSearchCode:='pack codes DB Error',
															sFssSendCode:='Validation_BadDB');

	stOuterBarcodeDBError:				ST_RejectItems :=(	nRejectID := 217,
															sMetsDisplayCode:= 'Outer code not found  - DB Error',
															sMetsSearchCode:='Outer code DB Error',
															sFssSendCode:='Validation_BadDB');

	stOuterCodesBrandSpecError	:		ST_RejectItems :=(	nRejectID := 218,
														sMetsDisplayCode:='Outer code invalid Brand',
														sMetsSearchCode:='Outer code invalid Brand',
														sFssSendCode:='Validation_BadCode');


	stUnknownOuterReject:		ST_RejectItems :=(	nRejectID := 200,
															sMetsDisplayCode:='',
															sMetsSearchCode:='',
															sFssSendCode:='UnknownReason');

END_STRUCT
END_TYPE

// ---- Data types/METS/AI Codes And Validation/ST_RejectReasonsForPack.TcDUT
TYPE ST_RejectReasonsForPack :
STRUCT
	stPackCodesNotLinked:		ST_RejectItems :=(	nRejectID := 101,
														sMetsDisplayCode:='Pack code(s) not linked',
														sMetsSearchCode:='Pack code(s) not linked',
														sFssSendCode:='NoPackData');

	stPackCodesOverwritten:		ST_RejectItems :=(	nRejectID := 102,
														sMetsDisplayCode:='Pack code(s) over-written',
														sMetsSearchCode:='Pack code(s) over-written',
														sFssSendCode:='WrongReadPackCode');

	stPackCodesGtinError:		ST_RejectItems :=(	nRejectID := 103,
														sMetsDisplayCode:='Pack code(s) invalid GTIN',
														sMetsSearchCode:='Pack code(s) invalid GTIN',
														sFssSendCode:='WrongMasterData');

	stPackCodesSerialError:		ST_RejectItems :=(	nRejectID := 104,
														sMetsDisplayCode:='Pack code(s) invalid Serial Code',
														sMetsSearchCode:='Pack code(s) invalid Serial Code',
														sFssSendCode:='Validation_BadCode');

	stPackCodeInvalidLength	:	ST_RejectItems :=(	nRejectID := 105,
														sMetsDisplayCode:='Pack code(s) invalid Length',
														sMetsSearchCode:='Pack code(s) invalid Length',
														sFssSendCode:='Validation_BadCode');

	stPackCodesNotRead:		ST_RejectItems :=(	nRejectID := 106,
														sMetsDisplayCode:='Pack code(s) no read',
														sMetsSearchCode:='Pack code(s) no read',
														sFssSendCode:='NoReadPackCode');

	stPackCodesDuplicated:		ST_RejectItems :=(	nRejectID := 107,
														sMetsDisplayCode:='Pack code(s) duplicate',
														sMetsSearchCode:='Pack code(s) duplicate',
														sFssSendCode:='Validation_BadCode');

	stPackCodesTypeError:		ST_RejectItems :=(	nRejectID := 108,
														sMetsDisplayCode:='Pack code(s) invalid type',
														sMetsSearchCode:='Pack code(s) invalid type',
														sFssSendCode:='Validation_BadType');

	stPackCodesSUPIError:		ST_RejectItems :=(	nRejectID := 109,
														sMetsDisplayCode:='Pack code(s) SUPI failed validation',
														sMetsSearchCode:='Pack code(s) SUPI failed validation',
														sFssSendCode:='Validation_BadSUPI');


	stPackCodesDBError:		ST_RejectItems :=(	nRejectID := 110,
														sMetsDisplayCode:='Pack code DB failed validation',
														sMetsSearchCode:='Pack code DB failed validation',
														sFssSendCode:='Validation_BadDB');

	stPackCodesBrandSpec:		ST_RejectItems :=(	nRejectID := 111,
														sMetsDisplayCode:='Pack code(s) invalid Brand',
														sMetsSearchCode:='Pack code(s) invalid Brand',
														sFssSendCode:='Validation_BadCode');


	stUnknownPackReject:		ST_RejectItems :=(	nRejectID := 100,
														sMetsDisplayCode:='UnknownReason',
														sMetsSearchCode:='UnknownReason',
														sFssSendCode:='UnknownReason');


END_STRUCT
END_TYPE

// ---- Data types/METS/Alarms/E_MessageID.TcDUT
{attribute 'qualified_only'}
{attribute 'to_string'}
TYPE E_MessageID :
(
	MSG_000 := 0,
	MSG_001,
	MSG_002,
	MSG_003,
	MSG_004,
	MSG_005,
	MSG_006,
	MSG_007,
	MSG_008,
	MSG_009,
	MSG_010,
	MSG_011,
	MSG_012,
	MSG_013,
	MSG_014,
	MSG_015,
	MSG_016,
	MSG_017,
	MSG_018,
	MSG_019,
	MSG_020,
	MSG_021,
	MSG_022,
	MSG_023,
	MSG_024,
	MSG_025,
	MSG_026,
	MSG_027,
	MSG_028,
	MSG_029,
	MSG_030,
	MSG_031,
	MSG_032,
	MSG_033,
	MSG_034,
	MSG_035,
	MSG_036,
	MSG_037,
	MSG_038,
	MSG_039,
	MSG_040,
	MSG_041,
	MSG_042,
	MSG_043,
	MSG_044,
	MSG_045,
	MSG_046,
	MSG_047,
	MSG_048,
	MSG_049,
	MSG_050,
	MSG_051,
	MSG_052,
	MSG_053,
	MSG_054,
	MSG_055,
	MSG_056,
	MSG_057,
	MSG_058,
	MSG_059,
	MSG_060,
	MSG_061,
	MSG_062,
	MSG_063,
	MSG_064,
	MSG_065,
	MSG_066,
	MSG_067,
	MSG_068,
	MSG_069,
	MSG_070,
	MSG_071,
	MSG_072,
	MSG_073,
	MSG_074,
	MSG_075,
	MSG_076,
	MSG_077,
	MSG_078,
	MSG_079,
	MSG_080,
	MSG_081,
	MSG_082,
	MSG_083,
	MSG_084,
	MSG_085,
	MSG_086,
	MSG_087,
	MSG_088,
	MSG_089,
	MSG_090,
	MSG_091,
	MSG_092,
	MSG_093,
	MSG_094,
	MSG_095,
	MSG_096,
	MSG_097,
	MSG_098,
	MSG_099,
	MSG_100,
	MSG_101,
	MSG_102,
	MSG_103,
	MSG_104,
	MSG_105,
	MSG_106,
	MSG_107,
	MSG_108,
	MSG_109,
	MSG_110,
	MSG_111,
	MSG_112,
	MSG_113,
	MSG_114,
	MSG_115,
	MSG_116,
	MSG_117,
	MSG_118,
	MSG_119,
	MSG_120,
	MSG_121,
	MSG_122,
	MSG_123,
	MSG_124,
	MSG_125,
	MSG_126,
	MSG_127,
	MSG_128,
	MSG_129,
	MSG_130,
	MSG_131,
	MSG_132,
	MSG_133,
	MSG_134,
	MSG_135,
	MSG_136,
	MSG_137,
	MSG_138,
	MSG_139,
	MSG_140,
	MSG_141,
	MSG_142,
	MSG_143,
	MSG_144,
	MSG_145,
	MSG_146,
	MSG_147,
	MSG_148,
	MSG_149,
	MSG_150,
	MSG_151,
	MSG_152,
	MSG_153,
	MSG_154,
	MSG_155,
	MSG_156,
	MSG_157,
	MSG_158,
	MSG_159,
	MSG_160,
	MSG_161,
	MSG_162,
	MSG_163,
	MSG_164,
	MSG_165,
	MSG_166,
	MSG_167,
	MSG_168,
	MSG_169,
	MSG_170,
	MSG_171,
	MSG_172,
	MSG_173,
	MSG_174,
	MSG_175,
	MSG_176,
	MSG_177,
	MSG_178,
	MSG_179,
	MSG_180,
	MSG_181,
	MSG_182,
	MSG_183,
	MSG_184,
	MSG_185,
	MSG_186,
	MSG_187,
	MSG_188,
	MSG_189,
	MSG_190,
	MSG_191,
	MSG_192,
	MSG_193,
	MSG_194,
	MSG_195,
	MSG_196,
	MSG_197,
	MSG_198,
	MSG_199,
	MSG_200,
	MSG_201,
	MSG_202,
	MSG_203,
	MSG_204,
	MSG_205,
	MSG_206,
	MSG_207,
	MSG_208,
	MSG_209,
	MSG_210,
	MSG_211,
	MSG_212,
	MSG_213,
	MSG_214,
	MSG_215,
	MSG_216,
	MSG_217,
	MSG_218,
	MSG_219,
	MSG_220,
	MSG_221,
	MSG_222,
	MSG_223,
	MSG_224,
	MSG_225,
	MSG_226,
	MSG_227,
	MSG_228,
	MSG_229,
	MSG_230,
	MSG_231,
	MSG_232,
	MSG_233,
	MSG_234,
	MSG_235,
	MSG_236,
	MSG_237,
	MSG_238,
	MSG_239,
	MSG_240,
	MSG_241,
	MSG_242,
	MSG_243,
	MSG_244,
	MSG_245,
	MSG_246,
	MSG_247,
	MSG_248,
	MSG_249,
	MSG_250,
	MSG_251,
	MSG_252,
	MSG_253,
	MSG_254,
	MSG_255
);
END_TYPE

// ---- Data types/METS/Alarms/ST_Alarms.TcDUT
TYPE ST_Alarms :
STRUCT
	nMessage						: 	DWORD;
	//nMessageTimer				:	ARRAY[0..31] OF TON;
	//nCategory					:	ARRAY[0..31] OF INT;
	nMessageType					:	WORD;
END_STRUCT
END_TYPE

// ---- Data types/METS/Alarms/ST_AlarmSettings.TcDUT
TYPE ST_AlarmSettings :
STRUCT
	aTextMessageTable		: ARRAY [0..31] OF STRING(200);
	aAlarmTriggerTable		: ARRAY [0..31] OF BOOL;

	aAlarmTimoutTable		: ARRAY [0..31] OF TIME;
	aBlockEnableTable			: ARRAY [0..31] OF BOOL :=[ 32 (FALSE)];
	aInhibitResetTable			: ARRAY [0..31] OF BOOL;
	aAutoResetTable			: ARRAY[0..31] OF BOOL;
	aInternalResetTable		: ARRAY [0..31] OF BOOL;

	aCategoryNoTable			: ARRAY[0..31] OF INT;
	aMessageTypeStatusTable	: ARRAY[0..31] OF WORD;
END_STRUCT
END_TYPE

// ---- Data types/METS/Alarms/ST_AlarmsTable.TcDUT
TYPE ST_AlarmsTable :
STRUCT
	//aTextMessages	 					: 	ARRAY [0..cMAX_MESSAGE_NUMBER] OF STRING(200);
	aActiveID							: 	ARRAY [0..cMAX_MESSAGE_NUMBER] OF BOOL;
	//aDisableAlarmLog					:	ARRAY [0..cMAX_MESSAGE_NUMBER] OF BOOL;


	aMsgHMI							:	ARRAY [0..cMAX_MESSAGE_NUMBER] OF T_MaxString;
	//aAlarmDB							:	ARRAY [0..cMAX_MESSAGE_NUMBER] OF ST_AlarmDB;
	aMsgAux							:	ARRAY [0..cMAX_MESSAGE_NUMBER] OF ST_ALARM_Aux;
	
	aLogMessages						:	ARRAY[1..cMAX_DISPLAY_ALARMS] OF STRING(200);
	aActiveMessages					:	ARRAY[1..15] OF STRING(200);
	
	aActiveMessagesHMI				:	ARRAY[1..15] OF INT:=[ 15(-1)];

	aLogDateAlarmsHMI				:	ARRAY[1..cMAX_DISPLAY_ALARMS] OF STRING(19);	(* date/time as HH:MM:SS DD/MM/YYYY for HMI display *)
	aLogAlarmsHMI					:	ARRAY[1..cMAX_DISPLAY_ALARMS] OF INT :=[ cMAX_DISPLAY_ALARMS(-1)];
	
	aLogDateWarningsHMI				:	ARRAY[1..cMAX_DISPLAY_ALARMS] OF STRING(19);	(* date/time as HH:MM:SS DD/MM/YYYY for HMI display *)
	aLogWarningsHMI					:	ARRAY[1..cMAX_DISPLAY_ALARMS] OF INT :=[ cMAX_DISPLAY_ALARMS(-1)];


END_STRUCT
END_TYPE

// ---- Data types/METS/Alarms/ST_AlarmStatus.TcDUT
TYPE ST_AlarmStatus :
STRUCT
	bNoActiveAlarms					: BOOL;
	bNoActiveWarrnings				: BOOL;

	bGeneralSystemAlarmActive		: BOOL;		(*Message type 0*)
	bEUCASubsytemAlarmActive		: BOOL;		(*Message type 1*)
	bTPDSubsytemAlarmActive		: BOOL;		(*Message type 2*)
	bExternalAlarmActive				: BOOL;		(*Message type 3*)

	bSpare04AlarmActive				: BOOL;		(*Message type 4*)
	bSpare05AlarmActive				: BOOL;		(*Message type 5*)
	bSpare06AlarmActive				: BOOL;		(*Message type 6*)
	bSpare07AlarmActive				: BOOL;		(*Message type 7*)

	bGeneralSystemWarningActive		: BOOL;		(*Message type 8*)
	bEUCASubsytemWarningActive	: BOOL;		(*Message type 9*)
	bTPDSubsytemWarningActive		: BOOL;		(*Message type 10*)
	bExternalWarningActive			: BOOL;		(*Message type 11*)

	bSpare12WarningActive			: BOOL;		(*Message type 12*)
	bSpare13WarningActive			: BOOL;		(*Message type 13*)
	bSpare14WarningActive			: BOOL;		(*Message type 14*)
	bSpare15WarningActive			: BOOL;		(*Message type 15*)

	(*eMessageType					: E_MessageType;*)
END_STRUCT
END_TYPE

// ---- Data types/METS/Alarms/ST_ALARM_Aux.TcDUT
TYPE ST_ALARM_Aux :
STRUCT
	nCategoryNo	: INT;
	nMessageTypeNo	: INT;
	sTextMessage	: STRING;
	bAutoReset		: BOOL;
END_STRUCT
END_TYPE

// ---- Data types/METS/Aliases/T_CAC_Filename.TcDUT
TYPE T_CAC_Filename : T_MaxString;
END_TYPE

// ---- Data types/METS/Aliases/T_CASE_Barcode.TcDUT
TYPE T_CASE_Barcode : T_MaxString;
END_TYPE

// ---- Data types/METS/Aliases/T_Char.TcDUT
TYPE T_Char : STRING[1];
END_TYPE

// ---- Data types/METS/Aliases/T_CHM_Filename.TcDUT
TYPE T_CHM_Filename : T_MaxString;
END_TYPE

// ---- Data types/METS/Aliases/T_CodeBATCH.TcDUT
 TYPE T_CodeBATCH : STRING[10];
END_TYPE

// ---- Data types/METS/Aliases/T_CodeBRAND.TcDUT
 TYPE T_CodeBRAND : STRING[9];
END_TYPE

// ---- Data types/METS/Aliases/T_CodeCRYPTO.TcDUT
TYPE T_CodeCRYPTO : STRING[20];
END_TYPE

// ---- Data types/METS/Aliases/T_CodeMRP.TcDUT
TYPE T_CodeMRP : STRING[8];
END_TYPE

// ---- Data types/METS/Aliases/T_CodePIT.TcDUT
TYPE T_CodePIT : STRING[7];
END_TYPE

// ---- Data types/METS/Aliases/T_CodePO.TcDUT
TYPE T_CodePO : STRING[20];
END_TYPE

// ---- Data types/METS/Aliases/T_CodePRODUCEDATE.TcDUT
 TYPE T_CodePRODUCEDATE : STRING[14];
END_TYPE

// ---- Data types/METS/Aliases/T_CodeRSKU.TcDUT
 TYPE T_CodeRSKU : STRING[9];
END_TYPE

// ---- Data types/METS/Aliases/T_CodeURL.TcDUT
TYPE T_CodeURL : STRING[20];
END_TYPE

// ---- Data types/METS/Aliases/T_DB_LongSTRING.TcDUT
TYPE T_DB_LongSTRING : STRING(1024);
END_TYPE

// ---- Data types/METS/Aliases/T_FileExtension.TcDUT
TYPE T_FileExtension : STRING[4];
END_TYPE

// ---- Data types/METS/Aliases/T_FolderName.TcDUT
TYPE T_FolderName : STRING[25];
END_TYPE

// ---- Data types/METS/Aliases/T_FSS_RejecCode.TcDUT
TYPE T_FSS_RejecCode : STRING(40);
END_TYPE

// ---- Data types/METS/Aliases/T_HMI_PACK_Barcode.TcDUT
TYPE T_HMI_PACK_Barcode : STRING(cMAX_HMI_PACKCODE_LENGHT);
END_TYPE

// ---- Data types/METS/Aliases/T_ISO8601Time.TcDUT
TYPE T_ISO8601Time : STRING(30);
END_TYPE

// ---- Data types/METS/Aliases/T_LongSTRING.TcDUT
TYPE T_LongSTRING : STRING(1023);
END_TYPE

// ---- Data types/METS/Aliases/T_OAC_Filename.TcDUT
TYPE T_OAC_Filename : T_MaxString;
END_TYPE

// ---- Data types/METS/Aliases/T_OCV_Filename.TcDUT
TYPE T_OCV_Filename : T_MaxString;
END_TYPE

// ---- Data types/METS/Aliases/T_OHM_Filename.TcDUT
TYPE T_OHM_Filename : STRING(44);
END_TYPE

// ---- Data types/METS/Aliases/T_OUTER_Barcode.TcDUT
TYPE T_OUTER_Barcode : T_MaxString;
END_TYPE

// ---- Data types/METS/Aliases/T_PACK_Barcode.TcDUT
TYPE T_PACK_Barcode : STRING(cMAX_PACKCODE_LENGHT);
END_TYPE

// ---- Data types/METS/Aliases/T_PCM_Filename.TcDUT
 TYPE T_PCM_Filename : T_MaxString;
END_TYPE

// ---- Data types/METS/Aliases/T_ProductDescription.TcDUT
TYPE T_ProductDescription : STRING[48];
END_TYPE

// ---- Data types/METS/Aliases/T_RejectCode.TcDUT
TYPE T_RejectCode : STRING[100];
END_TYPE

// ---- Data types/METS/Aliases/T_TimeLog.TcDUT
TYPE T_TimeLog : STRING[15];
END_TYPE

// ---- Data types/METS/Case/CAC/E_CAC_State.TcDUT
TYPE E_CAC_State :
(
	E_CAC_IDLE,
	E_CAC_OPENFILE,
	E_CAC_BUILDXMLIMAGE,
	E_CAC_WRITEXMLIMAGE,
	E_CAC_CLOSEXMLIMAGE,
	E_CAC_CLOSEFILE,
	E_CAC_FINDFOLDER,
	E_CAC_FINDFILE,
	E_CAC_READDATA,
	E_CAC_WRITEDATA,
	E_CAC_CREATEFOLDER,
	E_CAC_DELETEFOLDER,
	E_CAC_DELETEFILE,
	E_CAC_CREATEOACDATA,
	E_CAC_CREATEOCVDATA,
	E_CAC_WRITEOCVDATA,
	E_CAC_DELETEOAC,
	E_CAC_DELETEOCV1,
	E_CAC_DELETEOCV2,
	E_CAC_COPYFILE,
	E_CAC_MOVEFILE,
	E_CAC_RENAMEFILE,
	E_CAC_VALIDATECASE,
	E_CAC_VALIDATEOUTER,
	E_CAC_VALIDATEOAC,
	E_CAC_VALIDATEPACK,
	E_CAC_DUPLICATEOUTERCHECK,
	E_CAC_DBREQUEST,
	E_CAC_DBRESPONSE,
	E_CAC_CHECKOUTERDUPLICATES,
	E_CAC_CHECKPACKDUPLICATES,
	E_CAC_DONE
);
END_TYPE

// ---- Data types/METS/Case/CAC/ST_CAC_Data.TcDUT
TYPE ST_CAC_Data :
STRUCT
	Barcode 					: T_CASE_Barcode;
	ProductionDate			: STRING(10);
	ProductionTime			: STRING(8);
	ProductionTimeOffset		: STRING(6);		(* time offset between system and UTC, '+1:00' means SystemTime = UTC + 1hr *)
	RetailSKU					: T_CodeRSKU;
	CasePacker				: ST_SYSTEM_MachineID;
	CodingAndTrackingMode		: INT;
	NumberOfOuters			: INT;
	CaseRejectCode			: T_RejectCode; (* blank and not included in CAC files for valid cases *)
	CaseRejectID				: UINT	; (* blank and not included in CAC files for valid cases *)
	Outer					: ARRAY[1..cMAX_OUTERS_PER_CASE] OF ST_OAC_Data;
END_STRUCT
END_TYPE

// ---- Data types/METS/Case/CHM/CHM Data Structure/ST_Attributes.TcDUT
TYPE ST_Attributes :
STRUCT

	ProduceDateMC			: STRING(14);

END_STRUCT
END_TYPE

// ---- Data types/METS/Case/CHM/CHM Data Structure/ST_CHM_GenericHierarchy.TcDUT
TYPE ST_CHM_GenericHierarchy :
STRUCT
	HierarchyType		:	STRING(5);
	PerformedAction	:	STRING(10);
	TrackingLevels		:	STRING(10);
	TrackingIndicator	:	STRING(3);
	CaseItem			:	ST_CaseItem;

END_STRUCT
END_TYPE

// ---- Data types/METS/Case/CHM/CHM Data Structure/ST_GenericHierarchy.TcDUT
TYPE ST_GenericHierarchy :
STRUCT
	HierarchyType		:	STRING(5);
	PerformedAction	:	STRING(10);
	TrackingLevels		:	STRING(10);
	TrackingIndicator	:	STRING(3);
	CaseItem			:	ST_CaseItem;

END_STRUCT
END_TYPE

// ---- Data types/METS/Case/CHM/CHM Data Structure/ST_MessageHeader.TcDUT
TYPE ST_MessageHeader :
STRUCT

	(*CreationDate 				: STRING(10);
	CreationTime 				: STRING(25);*)
	ReferenceID				: T_MaxString;
	CreationTimeLocalUTC		: T_ISO8601Time;
	MessageType	 			: STRING(25);
	SenderSystem				: STRING(5);
	ReceiverSystem			: STRING(5);


END_STRUCT
END_TYPE

// ---- Data types/METS/Case/CHM/E_CHM_GeneratorState.TcDUT
TYPE E_CHM_GeneratorState :
(
	E_CHM_IDLEGENERATOR,
	E_CHM_FILECHECK,
	E_CHM_FILEOPEN,
	E_CHM_GENERATEHEAD,
	(*E_CHM_HEADDONE,*)
	E_CHM_GENERATEBODY,
	(*E_CHM_BODYDONE,*)
	E_CHM_GENERATEENDING,
	(*E_CHM_ENDINGDONE,*)
	E_CHM_FILECLOSE,
	E_CHM_GENERATEFLG,
	(*E_CHM_FLGDONE,*)
	E_CHM_TIMEOUT,
	E_CHM_DONEGENERATOR
);
END_TYPE

// ---- Data types/METS/Case/CHM/E_CHM_State.TcDUT
TYPE E_CHM_State :
(
	E_CHM_IDLE,
	E_CHM_OPENFILE,
	E_CHM_BUILDXMLIMAGE,
	E_CHM_WRITEXMLIMAGE,
	E_CHM_CLOSEFILE,
	E_CHM_FINDFOLDER,
	E_CHM_FINDFILE,
	E_CHM_READDATA,
	E_CHM_WRITEDATA,
	E_CHM_CREATEFOLDER,
	E_CHM_DELETEFOLDER,
	E_CHM_DELETEFILE,
	E_CHM_COPYFILE,
	E_CHM_MOVEFILE,
	E_CHM_RENAMEFILE,
	E_CHM_VALIDATECASE,
	E_CHM_VALIDATEOUTER,
	E_CHM_VALIDATEOAC,
	E_CHM_VALIDATEPACK,
	E_CHM_DUPLICATEOUTERCHECK,
	E_CHM_DONE
);
END_TYPE

// ---- Data types/METS/Case/CHM/E_CHM_WriteMode.TcDUT
TYPE E_CHM_WriteMode :
(
	E_CHM_FSS2MODE_NOBACKUP,
	E_CHM_FSS2MODE_FSS2BACKUP,
	E_CHM_FSS3MODE_NOBACKUP,
	E_CHM_FSS3MODE_FSS2BACKUP

);
END_TYPE

// ---- Data types/METS/Case/CHM/ST_CHM_Data.TcDUT
TYPE ST_CHM_Data :
STRUCT
	MessageHeader		:	ST_MessageHeader;
	Factory				:	STRING(3);
	GenericHierarchy		:	ST_GenericHierarchy;
	Attributes				:	ST_Attributes;
END_STRUCT
END_TYPE

// ---- Data types/METS/Case/E_CASE_State.TcDUT
TYPE E_CASE_State :
(
	E_CASE_IDLE,
	E_CASE_SCANINFEEDQUEUE,
	E_CASE_COPYOACFILE,
	E_CASE_READOACDATA,
	E_CASE_SCANOUTERS,
	E_CASE_DUPLICATEPACKCHECK,
	E_CASE_UPDATEINFEEDQUEUE,
	E_CASE_DELETEOACFILE,
	E_CASE_DELETEOCV1FILE,
	E_CASE_DELETEOCV2FILE,
	E_CASE_VALIDATECAC,
	E_CASE_GETSERIALCODE,
	E_CASE_FINDCACFILE,
	E_CASE_RENAMECACFILE,
	E_CASE_MOVECACFILE,
	E_CASE_DATAVALIDATE,
	E_CASE_DATAWRITEXML,
	E_CASE_OVERWIRTECAC,
	E_CASE_DATAFINALISE,
	E_CASE_DONE
);
END_TYPE

// ---- Data types/METS/Case/ORCA/E_ORCA_State.TcDUT
TYPE E_ORCA_State :
(
	E_ORCA_IDLE,
	E_ORCA_OPENFILE,

	E_ORCA_CLOSEFILE,
	E_ORCA_FINDFOLDER,
	E_ORCA_FINDFILE,
	E_ORCA_READDATA,

	E_ORCA_DELETEFILE,
	E_ORCA_COPYFILE,
	E_ORCA_MOVEFILE,
	E_ORCA_RENAMEFILE,

	E_ORCA_VALIDATEOUTER,
	E_ORCA_VALIDATEOAC,

	E_ORCA_DONE
);
END_TYPE

// ---- Data types/METS/Case/ORCA/ST_ORCA_BrandInfo.TcDUT
TYPE ST_ORCA_BrandInfo :
STRUCT

	BatchID 			: STRING(255);
	GTIN 			: STRING(255);
	SKU 				: STRING(255);
	ProductionOrder 	: STRING(255);

END_STRUCT
END_TYPE

// ---- Data types/METS/Case/ORCA/ST_ORCA_Data.TcDUT
TYPE ST_ORCA_Data :
STRUCT
	SiteInfo 				: ST_ORCA_SiteInfo;
	BrandInfo 			: ST_ORCA_BrandInfo;
	ProductInfo			: ST_ORCA_ProductInfo;
	Outers				: ARRAY[1..60] OF ST_ORCA_Outers;

END_STRUCT
END_TYPE

// ---- Data types/METS/Case/ORCA/ST_ORCA_Outers.TcDUT
TYPE ST_ORCA_Outers :
STRUCT
	Code 	: STRING(255);
	xPos		: INT;
	yPos		: INT;

END_STRUCT
END_TYPE

// ---- Data types/METS/Case/ORCA/ST_ORCA_ProductInfo.TcDUT
TYPE ST_ORCA_ProductInfo :
STRUCT

	OutersPerRow 			: STRING(255);
	RowsPerCase	 		: STRING(255);


END_STRUCT
END_TYPE

// ---- Data types/METS/Case/ORCA/ST_ORCA_SiteInfo.TcDUT
TYPE ST_ORCA_SiteInfo :
STRUCT

	ProductionSite 			: STRING(255);
	ProductionLine 		: STRING(255);


END_STRUCT
END_TYPE

// ---- Data types/METS/Case/ST_CasePackerInfo.TcDUT
TYPE ST_CasePackerInfo :	(* 8 bytes *)
STRUCT
	ProductionSite 	: STRING(4);
	ProductionLine 	: STRING(4);
END_STRUCT
END_TYPE

// ---- Data types/METS/Case/ST_CASE_CaseQueue.TcDUT
TYPE ST_CASE_CaseQueue :
STRUCT
	aCACData		: ARRAY[1..cMAX_CASE_QUEUE] OF ST_CAC_Data;	(* array of CAC data *)
	stPrintCACData	: ST_CAC_Data;	(* CAC data sent to printer *)

	stPrintCHMData	: ST_CHM_Data;	(* CHM data printed to XML file *)
END_STRUCT
END_TYPE

// ---- Data types/METS/Case/ST_CASE_DefferOuter.TcDUT
TYPE ST_CASE_DefferOuter :
STRUCT
	sID 					: STRING(255);
	ProductionDate 		: STRING(10);
	ProductionTime 		: STRING(8);
	ProductionTimeOffset 	: STRING(6);
	RejectCode 			: STRING(255);
END_STRUCT
END_TYPE

// ---- Data types/METS/Case/ST_CASE_OperationData.TcDUT
TYPE ST_CASE_OperationData :
STRUCT

	nActualNumberOfOutersIndex		: UINT;
	nFianalNumberOfOutersIndex		: INT;
	nCrossPushToCaseIndex			: UINT;

	nAcceptedWeight					: UDINT;
	nRejectedWeight					: UDINT;
		
	bDoorOpen						: BOOL;
	
	bCheckDuplicates				: BOOL;
	bIsDuplicateOuters				: BOOL;
	bIsDuplicatePacks				: BOOL;

	bReadyToValidate				: BOOL;
	nValidationIndex				: INT;
	nMasterListRestoreIndex			: INT;

	bCaseAccepted					: BOOL;
	bCaseRejected					: BOOL;

	sValidateRejectCode				: T_MaxString;
	nValidationErrorID 				: UINT;

	sFirstBarcodeInCase				: T_OUTER_Barcode;
	sLastBarcodeInCase				: T_OUTER_Barcode;


END_STRUCT
END_TYPE

// ---- Data types/METS/Device/CX Unit/EtherCAT/E_CX_EtherCATState.TcDUT
{attribute 'qualified_only'}
{attribute 'strict'}
TYPE E_CX_EtherCATState : (
	IDLE,
	READADDR,
	READSTATE,
	MAP,
	//E_CX_ETHERCAT_IORESET,
	//E_CX_ETHERCAT_SETINITMODE,
	//E_CX_ETHERCAT_WAITINITMODE,
	//E_CX_ETHERCAT_SETOPMODE,
	//E_CX_ETHERCAT_WAITOPMODE,
	DONE
);
END_TYPE

// ---- Data types/METS/Device/CX Unit/EtherCAT/ST_CX_EtherCATDeviceState.TcDUT
TYPE ST_CX_EtherCATDeviceState :
STRUCT
	bPresent		: BOOL;
	bOpMode			: BOOL;
	bError			: BOOL;
	nDeviceState	: BYTE;
	nLinkState		: BYTE;
	strStatus		: STRING(17);
END_STRUCT
END_TYPE

// ---- Data types/METS/Device/CX Unit/EtherCAT/ST_CX_EtherCATMasterPNetState.TcDUT
TYPE ST_CX_EtherCATMasterPNetState :
STRUCT
	arrADSAddr		: ARRAY[0..5] OF BYTE;
	nPortNo			: UINT;
	arrAoeAddr		: ARRAY[0..5] OF BYTE;
	nDevState		: UINT;
	nPnIoError		: UINT;
	nPnIoDiag			: UINT;
END_STRUCT
END_TYPE

// ---- Data types/METS/Device/CX Unit/EtherCAT/ST_CX_EtherCATMasterState.TcDUT
TYPE ST_CX_EtherCATMasterState :
STRUCT
	arrADSAddr		: ARRAY[0..5] OF BYTE;
	nState			: UINT;
	nDevID			: UINT;
	nSlaveCount		: UINT;
	nDevState		: UINT;
END_STRUCT
END_TYPE

// ---- Data types/METS/Device/CX Unit/Network/ST_CX_AdapterInfo.TcDUT
TYPE ST_CX_AdapterInfo :
STRUCT
	bDefault			: BOOL;
	strAdapterName		: STRING(75);
	bDHCPEnabled		: BOOL;
	strIPAddress		: T_IPv4Addr;
	strSubnetMask		: T_IPv4Addr;
	strDefaultGateway	: T_IPv4Addr;
END_STRUCT
END_TYPE

// ---- Data types/METS/Device/CX Unit/Network/ST_CX_NetworkInfo.TcDUT
TYPE ST_CX_NetworkInfo :
STRUCT
	strDeviceName		: STRING(75);
	strAMSNetID			: STRING(23);
	strSNTPServer		: STRING(75);
	strSNTPRefreshTime	: STRING(31);
	arrAdapterInfo		: ARRAY[1..6] OF ST_CX_AdapterInfo;
END_STRUCT
END_TYPE

// ---- Data types/METS/Device/CX Unit/NOVRAM/E_CX_NVDataOpMode.TcDUT
{attribute 'qualified_only'}
{attribute 'strict'}
TYPE E_CX_NVDataOpMode : (
	//E_CX_NVDATA_OPMODE_IDLE,
	//E_CX_NVDATA_OPMODE_EL6080,
	//E_CX_NVDATA_OPMODE_NOVRAM,
	//E_CX_NVDATA_OPMODE_BINARYFILE
	DUMMY
);
END_TYPE

// ---- Data types/METS/Device/CX Unit/NOVRAM/E_CX_NVXMLState.TcDUT
{attribute 'qualified_only'}
{attribute 'strict'}
TYPE E_CX_NVXMLState : (
	IDLE,
	READXML,
	RESTORE,
	MONITOR,
	WRITEXML,
	BACKUP,
	RETRY
);
END_TYPE

// ---- Data types/METS/Device/CX Unit/NOVRAM/ST_CX_AMSAddress.TcDUT
TYPE ST_CX_AMSAddress :
STRUCT
	arrAMSNetID			: AMSNETID;
	nPortNo				: UINT;
END_STRUCT
END_TYPE

// ---- Data types/METS/Device/CX Unit/NOVRAM/ST_CX_EL6080DataIn.TcDUT
TYPE ST_CX_EL6080DataIn :
STRUCT
	nStatus			: UINT;
	arrData			: ARRAY[0..1277] OF BYTE;
	bWcState		: BOOL;
	bInputToggle	: BOOL;
	nState			: UINT;
	sAMSAddress		: ST_CX_AMSAddress;
END_STRUCT
END_TYPE

// ---- Data types/METS/Device/CX Unit/NOVRAM/ST_CX_EL6080DataOut.TcDUT
TYPE ST_CX_EL6080DataOut :
STRUCT
	nControl		: UINT;
	arrData			: ARRAY[0..1277] OF BYTE;
END_STRUCT
END_TYPE

// ---- Data types/METS/Device/CX Unit/NOVRAM/ST_CX_NVDataBlock.TcDUT
TYPE ST_CX_NVDataBlock :
STRUCT
	DataOffs	: UDINT;
	Data		: STRING(2048);
END_STRUCT
END_TYPE

// ---- Data types/METS/Device/CX Unit/System/E_CX_State.TcDUT
{attribute 'qualified_only'}
{attribute 'strict'}
TYPE E_CX_State :
(
	IDLE,
	HW,
	OS,
	BASEFOLDER,
	DONE
);
END_TYPE

// ---- Data types/METS/Device/Cylinders/E_CYLINDER_Name.TcDUT
{attribute 'qualified_only'}
{attribute 'strict'}
TYPE E_CYLINDER_Name :
(
	CLAMP				:=1,
	GATE				:=2,
	REJECT				:=3,
	ADDITIONAL_REJECT	:=4,  {text 'change to ADDIT'}
	FIRST_PUSHER		:=5,
	SECOND_PUSHER		:=6

);
END_TYPE

// ---- Data types/METS/Device/Cylinders/ST_CYLINDER_Config.TcDUT
TYPE ST_CYLINDER_Config :
STRUCT

	bEnable					: BOOL;
	sDeviceName				: STRING(30) := 'Cylinder';
	tOperationalTime		: TIME := t#100ms;
	tTimeOut				: TIME := t#1s;
	bExtendAsHomePos	 	: BOOL;

	stTagID					: ST_CYLINDER_TagID;

END_STRUCT
END_TYPE

// ---- Data types/METS/Device/Cylinders/ST_CYLINDER_Control.TcDUT
TYPE ST_CYLINDER_Control :
STRUCT
	eCommand		: E_CYLINDER_Position;
END_STRUCT
END_TYPE

// ---- Data types/METS/Device/Cylinders/ST_CYLINDER_IN.TcDUT
TYPE ST_CYLINDER_IN :
STRUCT
	bEnable				: BOOL;
	bRelExtend			: BOOL;
	bRelRetract			: BOOL;
END_STRUCT
END_TYPE

// ---- Data types/METS/Device/Cylinders/ST_CYLINDER_Status.TcDUT
 TYPE ST_CYLINDER_Status :
STRUCT

	I					: ST_CYLINDER_IN;
	Q					: ST_CYLINDER_OUT;

END_STRUCT
END_TYPE

// ---- Data types/METS/Device/Cylinders/ST_CYLINDER_TagID.TcDUT
TYPE ST_CYLINDER_TagID :
STRUCT
	sDeviceTagID			: STRING(10);
	sRetractTagID			: STRING(10);
	sExtendTagID			: STRING(10);

END_STRUCT
END_TYPE

// ---- Data types/METS/Device/DB/E_DB_ScanState.TcDUT
(*
-------------------------------------------------------------------------------------------------
DATE		Version	Author	Comments
-------------------------------------------------------------------------------------------------
11/06/2020	1.00.00	CD		

-------------------------------------------------------------------------------------------------
*)
{attribute 'qualified_only'}
//{attribute 'strict'}
TYPE E_DB_ScanState :
(

	//E_DB_IDLE,
	//E_DB_SENDREQ,
	//E_DB_RECIVED,
	//E_DB_DONE
	DUMMY
);
END_TYPE

// ---- Data types/METS/Device/DB/OLD/ST_DBResult.TcDUT
TYPE ST_DBResult :
STRUCT
	strCode : STRING(150);
	nExpiryStatus : DINT;
	(*nNumberOfchildren : INT;*)

(* nExpiryStatus:
0 - Expired
1 - Unknown - probaly due to reanimation. should still be successful
2 - Not Expired - OK*)
END_STRUCT
END_TYPE

// ---- Data types/METS/Device/DB/OLD/ST_DB_CACCheckCtrl.TcDUT
TYPE ST_DB_CACCheckCtrl :
STRUCT
	bDB_ExecuteCacCheck			: BOOL;
	bDB_CACCheckComplete		: BOOL;
	bDB_CaseOk					: BOOL;
	bDB_Error						: BOOL;
	stCacToCheck					: ST_CAC_Data;
END_STRUCT
END_TYPE

// ---- Data types/METS/Device/DB/OLD/ST_DB_Config.TcDUT
TYPE ST_DB_Config :
STRUCT

	bDBConfigured				: BOOL;
	sSQLName					: STRING;
	sDatabaseName				: STRING;
	stNetAddress				: ST_TCPIP_AddressPort;
	nLastDBID					: UDINT;

	bEnableOCVCheck							: BOOL;
	bEnableOACCheck							: BOOL;
	bEnableCACCheck							: BOOL;

END_STRUCT
END_TYPE

// ---- Data types/METS/Device/DB/OLD/ST_DB_OACCheckCtrl.TcDUT
TYPE ST_DB_OACCheckCtrl :
STRUCT
	bDB_ExecuteOacCheck			: BOOL;
	bDB_OacCheckComplete			: BOOL;
	bOacValid						: BOOL;
	bDB_Error						: BOOL;
	stOacToCheck					: ST_OUTER_Status;
END_STRUCT
END_TYPE

// ---- Data types/METS/Device/DB/OLD/ST_DB_OCVCheckCtrl.TcDUT
TYPE ST_DB_OCVCheckCtrl :
STRUCT
	bDB_ExecuteOcvCheck			: BOOL;
	bDB_OcvCheckComplete			: BOOL;
	bDB_AllCodesFound				: BOOL;
	bDB_Error						: BOOL;
	bDB_OCVValid					: BOOL;
	stOcvToCheck 					: ST_OUTER_Status;
END_STRUCT
END_TYPE

// ---- Data types/METS/Device/DB/OLD/ST_DB_PcvCheckCtrl.TcDUT
TYPE ST_DB_PcvCheckCtrl :
STRUCT
	bDB_ExecutePcvCheck			: BOOL;
	bDB_PcvCheckComplete			: BOOL;
	bPackCodeFoundInDB			: BOOL;
	bPackExpired					: BOOL;
	sAssociatedCase 				: STRING(150);
	bDB_Error						: BOOL;
	stPackToCheck					: ST_PACK_Data;

END_STRUCT
END_TYPE

// ---- Data types/METS/Device/DB/OLD/ST_DB_ReportDBCtrl.TcDUT
TYPE ST_DB_ReportDBCtrl :
STRUCT
	bExecuteCheck			: BOOL;
	bCheckComplete			: BOOL;
	sStoreProcedureName		: STRING := 'TC_DBReport';
	bDBError				: BOOL;
	nDBErrorID				: UDINT;
	sSqlState				: ST_DBSQLError;
	nRecords				: UDINT;
	stResultRecord			: ST_DB_ReportResult;

END_STRUCT
END_TYPE

// ---- Data types/METS/Device/DB/OLD/ST_DB_ReportResult.TcDUT
TYPE ST_DB_ReportResult :
STRUCT
	nPackCodesTotal		: DINT;
	nPCV_NoDate 			: DINT;
	nPCV_NoOuterCode 	: DINT;
	nNoCACPack			: DINT;
	nOuterCodesTotal		: DINT;
	nOAC_NoDate 			: DINT;
	nNoOHMSuccesfull		: DINT;
	nNoCACOuter 			: DINT;
	nPackCodesArchive	 	: DINT;
	nOuterCodesArchive	: DINT;
END_STRUCT
END_TYPE

// ---- Data types/METS/Device/DB/ST_DB_CACDataCtrl.TcDUT
TYPE ST_DB_CACDataCtrl :
STRUCT
	bCreateDataReq				: BOOL;	(* C *)
	bReadDataReq				: BOOL;	(* R *)
	bUpdateDataReq				: BOOL;	(* U *)
	bDeleteDataReq				: BOOL;	(* D *)

	sFileCodeName				: T_MaxString;
	sArchiveName				: STRING;
		
	bBlockRecord				: BOOL;
	bReanimated					: BOOL;

	stCACStatusDB				: ST_CAC_Data;

	bDone						: BOOL;
	bError						: BOOL;
	nErrorID					: UDINT;


END_STRUCT
END_TYPE

// ---- Data types/METS/Device/Drive/Analog/ST_DriveCtrl.TcDUT
TYPE ST_DriveCtrl :
STRUCT
	bDriveRun:BOOL;
	nDriveAnalog:INT;
END_STRUCT
END_TYPE

// ---- Data types/METS/Device/Drive/Analog/ST_PhtcCtrl.TcDUT
TYPE ST_PhtcCtrl :
STRUCT
	bStopInfeedConveyor:BOOL;
	bStopSeparator:BOOL;
END_STRUCT
END_TYPE

// ---- Data types/METS/Device/Drive/MC2/E_MC_Name.TcDUT
{attribute 'qualified_only'}
{attribute 'strict'}
TYPE E_MC_Name :
(
	REVOLUTION		:=1	(*REVS*)
	//E_MC_SPARE	:=2	(*REVS*)
);
END_TYPE

// ---- Data types/METS/Device/Drive/Profinet/ST_PNetMasterStatus.TcDUT
TYPE ST_PNetMasterStatus :
(* EL6631 *)
STRUCT
	nPNetIoError		: UINT;
	nPNetIoDiag		: UINT;
END_STRUCT
END_TYPE

// ---- Data types/METS/Device/Encoders/CAMS/ST_AFS60_Cam.TcDUT
TYPE ST_AFS60_Cam :
STRUCT
	bEnable				: BOOL;
	nLowerLimit1		: UDINT;
	nLowerLimit2		: UDINT;
	nUpperLimit1		: UDINT;
	nUpperLimit2		: UDINT;
END_STRUCT
END_TYPE

// ---- Data types/METS/Device/Encoders/CAMS/ST_AFS60_CamHMi.TcDUT
TYPE ST_AFS60_CamHMi :
STRUCT
	bEnable				: BOOL;
	fLowerLimit1		: LREAL; (* channel 1 *)
	fLowerLimit2		: LREAL; (* channel 2 *)
	fUpperLimit1		: LREAL;
	fUpperLimit2		: LREAL;
	fRange				: LREAL := 360.0;
	sDesciption			: STRING := 'Cam';
END_STRUCT
END_TYPE

